HMI tags "2920RS001A01T02"
   "2920RS001A01T02.MSW" : 52809b66-421d-457f-8884-6f7a49d4e247 AT %DB5053.DBX18.0, 500 ms
   "2920RS001A01T02.DefaultText" : TextRef, internal   // Заголовок POPUP окна. При експорте из ECS через скрипт заполняется автоматически, если теги копируются в ручную то требуется в ручную задатать свойство Start Value
   "2920RS001A01T02.BlockInfo" : Array [0..2] of Int AT %DB5053.DBX38.0, 500 ms
   "2920RS001A01T02.StatusWork" : Int AT %DB5053.DBW242, 500 ms
   "2920RS001A01T02.FP_PARAM.DampingTime" : Int AT %DB5053.DBW50, 500 ms
   "2920RS001A01T02.FP_PARAM.Force_Value" : Real AT %DB5053.DBD52, 500 ms
   "2920RS001A01T02.FP_PARAM.Scale_Min" : Real AT %DB5053.DBD56, 500 ms
   "2920RS001A01T02.FP_PARAM.Scale_Max" : Real AT %DB5053.DBD60, 500 ms
   "2920RS001A01T02.FP_PARAM.Gradient" : Real AT %DB5053.DBD64, 500 ms
   "2920RS001A01T02.FP_PARAM.Grad_Pos" : Real AT %DB5053.DBD68, 500 ms
   "2920RS001A01T02.FP_PARAM.Grad_Neg" : Real AT %DB5053.DBD72, 500 ms
   "2920RS001A01T02.FP_PARAM.Grad_X" : Real AT %DB5053.DBD76, 500 ms
   "2920RS001A01T02.FP_PARAM.Gradient_Time_Pre" : Int AT %DB5053.DBW80, 500 ms
   "2920RS001A01T02.FP_PARAM.Gradient_Time_ACC" : Int AT %DB5053.DBW82, 500 ms
   "2920RS001A01T02.FP_PARAM.Alarm_Hyst" : Real AT %DB5053.DBD84, 500 ms
   "2920RS001A01T02.FP_PARAM.AlarmLimit_H3" : Real AT %DB5053.DBD88, 500 ms
   "2920RS001A01T02.FP_PARAM.AlarmLimit_H2" : Real AT %DB5053.DBD92, 500 ms
   "2920RS001A01T02.FP_PARAM.AlarmLimit_H1" : Real AT %DB5053.DBD96, 500 ms
   "2920RS001A01T02.FP_PARAM.AlarmLimit_L1" : Real AT %DB5053.DBD100, 500 ms
   "2920RS001A01T02.FP_PARAM.AlarmLimit_L2" : Real AT %DB5053.DBD104, 500 ms
   "2920RS001A01T02.FP_PARAM.AlarmLimit_L3" : Real AT %DB5053.DBD108, 500 ms
   "2920RS001A01T02.FP_PARAM.AlarmDelay_H3_Pre" : Int AT %DB5053.DBW112, 500 ms
   "2920RS001A01T02.FP_PARAM.AlarmDelay_H3_Acc" : Int AT %DB5053.DBW114, 500 ms
   "2920RS001A01T02.FP_PARAM.AlarmDelay_H2_Pre" : Int AT %DB5053.DBW116, 500 ms
   "2920RS001A01T02.FP_PARAM.AlarmDelay_H2_Acc" : Int AT %DB5053.DBW118, 500 ms
   "2920RS001A01T02.FP_PARAM.AlarmDelay_H1_Pre" : Int AT %DB5053.DBW120, 500 ms
   "2920RS001A01T02.FP_PARAM.AlarmDelay_H1_Acc" : Int AT %DB5053.DBW122, 500 ms
   "2920RS001A01T02.FP_PARAM.AlarmDelay_L1_Pre" : Int AT %DB5053.DBW124, 500 ms
   "2920RS001A01T02.FP_PARAM.AlarmDelay_L1_Acc" : Int AT %DB5053.DBW126, 500 ms
   "2920RS001A01T02.FP_PARAM.AlarmDelay_L2_Pre" : Int AT %DB5053.DBW128, 500 ms
   "2920RS001A01T02.FP_PARAM.AlarmDelay_L2_Acc" : Int AT %DB5053.DBW130, 500 ms
   "2920RS001A01T02.FP_PARAM.AlarmDelay_L3_Pre" : Int AT %DB5053.DBW132, 500 ms
   "2920RS001A01T02.FP_PARAM.AlarmDelay_L3_Acc" : Int AT %DB5053.DBW134, 500 ms
   "2920RS001A01T02.FP_PARAM.OpenLoopDelay_Pre" : Int AT %DB5053.DBW136, 500 ms
   "2920RS001A01T02.FP_PARAM.OpenLoopDelay_Acc" : Int AT %DB5053.DBW138, 500 ms
   "2920RS001A01T02.FP_PARAM.OverRangeDelay_Pre" : Int AT %DB5053.DBW140, 500 ms
   "2920RS001A01T02.FP_PARAM.OverRangeDelay_Acc" : Int AT %DB5053.DBW142, 500 ms
   "2920RS001A01T02.FP_PARAM.AuxLimit_H2_Value" : Real AT %DB5053.DBD144, 500 ms
   "2920RS001A01T02.FP_PARAM.AuxLimit_H1_Value" : Real AT %DB5053.DBD148, 500 ms
   "2920RS001A01T02.FP_PARAM.AuxLimit_L2_Value" : Real AT %DB5053.DBD152, 500 ms
   "2920RS001A01T02.FP_PARAM.AuxLimit_L1_Value" : Real AT %DB5053.DBD156, 500 ms
   "2920RS001A01T02.Unit" : TextRef, internal   // Еденицы измерения При експорте из ECS через скрипт заполняется автоматически, если теги копируются в ручную то требуется задатать свойство Text
   "2920RS001A01T02.Decimals" : TextRef, internal   // Формат отображения При експорте из ECS через скрипт, заполняется автоматически. Если теги копируются в ручную то требуется задатать свойство Text s999999.9
   "2920RS001A01T02.FP_EN.Square" : Bool AT %DB5053.DBX46.0, 500 ms
   "2920RS001A01T02.FP_EN.SquareRoot" : Bool AT %DB5053.DBX46.1, 500 ms
   "2920RS001A01T02.FP_EN.ParentSupress" : Bool AT %DB5053.DBX46.2, 500 ms
   "2920RS001A01T02.FP_EN.ParentSupressUnit" : Bool AT %DB5053.DBX46.3, 500 ms
   "2920RS001A01T02.FP_EN.Force" : Bool AT %DB5053.DBX46.4, 500 ms
   "2920RS001A01T02.FP_EN.Damping" : Bool AT %DB5053.DBX46.5, 500 ms
   "2920RS001A01T02.FP_EN.Gradient_Pos" : Bool AT %DB5053.DBX46.6, 500 ms
   "2920RS001A01T02.FP_EN.Gradient_Neg" : Bool AT %DB5053.DBX46.7, 500 ms
   "2920RS001A01T02.FP_EN.Hysteresis" : Bool AT %DB5053.DBX47.0, 500 ms
   "2920RS001A01T02.FP_EN.Alarm_H3" : Bool AT %DB5053.DBX47.1, 500 ms
   "2920RS001A01T02.FP_EN.Alarm_H2" : Bool AT %DB5053.DBX47.2, 500 ms
   "2920RS001A01T02.FP_EN.Alarm_H1" : Bool AT %DB5053.DBX47.3, 500 ms
   "2920RS001A01T02.FP_EN.Alarm_L1" : Bool AT %DB5053.DBX47.4, 500 ms
   "2920RS001A01T02.FP_EN.Alarm_L2" : Bool AT %DB5053.DBX47.5, 500 ms
   "2920RS001A01T02.FP_EN.Alarm_L3" : Bool AT %DB5053.DBX47.6, 500 ms
   "2920RS001A01T02.FP_EN.AlarmDelay_H3" : Bool AT %DB5053.DBX47.7, 500 ms
   "2920RS001A01T02.FP_EN.AlarmDelay_H2" : Bool AT %DB5053.DBX48.0, 500 ms
   "2920RS001A01T02.FP_EN.AlarmDelay_H1" : Bool AT %DB5053.DBX48.1, 500 ms
   "2920RS001A01T02.FP_EN.AlarmDelay_L1" : Bool AT %DB5053.DBX48.2, 500 ms
   "2920RS001A01T02.FP_EN.AlarmDelay_L2" : Bool AT %DB5053.DBX48.3, 500 ms
   "2920RS001A01T02.FP_EN.AlarmDelay_L3" : Bool AT %DB5053.DBX48.4, 500 ms
   "2920RS001A01T02.FP_EN.ROC_Warn" : Bool AT %DB5053.DBX48.5, 500 ms
   "2920RS001A01T02.FP_EN.U_Range_Warn" : Bool AT %DB5053.DBX48.6, 500 ms
   "2920RS001A01T02.FP_EN.O_Range_Warn" : Bool AT %DB5053.DBX48.7, 500 ms
   "2920RS001A01T02.trend_tag_name" : TextRef, internal   // Еденицы измерения При експорте из ECS через скрипт - заполняется автоматически, если теги копируются в ручную то требуется задатать свойство Text - имя тега для тренда
   "2920RS001A01T02.DQ.AL_H3" : Bool AT %DB5053.DBX16.0, 500 ms
   "2920RS001A01T02.DQ.AL_H2" : Bool AT %DB5053.DBX16.1, 500 ms
   "2920RS001A01T02.DQ.AL_H1" : Bool AT %DB5053.DBX16.2, 500 ms
   "2920RS001A01T02.DQ.AL_L1" : Bool AT %DB5053.DBX16.3, 500 ms
   "2920RS001A01T02.DQ.AL_L2" : Bool AT %DB5053.DBX16.4, 500 ms
   "2920RS001A01T02.DQ.AL_L3" : Bool AT %DB5053.DBX16.5, 500 ms
   "2920RS001A01T02.DQ.SIG_OK" : Bool AT %DB5053.DBX16.6, 500 ms
   "2920RS001A01T02.DQ.LIM_H2" : Bool AT %DB5053.DBX16.7, 500 ms
   "2920RS001A01T02.DQ.LIM_H1" : Bool AT %DB5053.DBX17.0, 500 ms
   "2920RS001A01T02.DQ.LIM_L1" : Bool AT %DB5053.DBX17.1, 500 ms
   "2920RS001A01T02.DQ.LIM_L2" : Bool AT %DB5053.DBX17.2, 500 ms
   "2920RS001A01T02.DQ.GR_P" : Bool AT %DB5053.DBX17.3, 500 ms
   "2920RS001A01T02.DQ.GR_N" : Bool AT %DB5053.DBX17.4, 500 ms
   "2920RS001A01T02.I.IN" : Real AT %DB5053.DBD2, 500 ms
   "2920RS001A01T02.I.SIG_TYPE" : Int AT %DB5053.DBW0, 500 ms
   "2920RS001A01T02.I.FI_BUS" : Byte AT %DB5053.DBB6, 500 ms
   "2920RS001A01T02.DI.U_RANGE" : Bool AT %DB5053.DBX7.0, 500 ms
   "2920RS001A01T02.DI.O_RANGE" : Bool AT %DB5053.DBX7.1, 500 ms
   "2920RS001A01T02.DI.SIG_FAULT" : Bool AT %DB5053.DBX7.2, 500 ms
   "2920RS001A01T02.DI.EnConfig" : Bool AT %DB5053.DBX7.3, 500 ms
   "2920RS001A01T02.DI.AEN" : Bool AT %DB5053.DBX7.4, 500 ms
   "2920RS001A01T02.DI.AL_SUPR" : Bool AT %DB5053.DBX7.5, 500 ms
   "2920RS001A01T02.Q.PV_NORM" : Real AT %DB5053.DBD8, 500 ms
   "2920RS001A01T02.Q.PV_SCAL" : Real AT %DB5053.DBD12, 500 ms
   "2920RS001A01T02.ParentInfo" : TextRef, internal   // Имя родителя для попап окна, вкладка инфо. При експорте из ECS через скрипт заполняется автоматически, если теги копируются в ручную то требуется в ручную задатать свойство Start Value

HMI tags "2920RS001A01T03"
   "2920RS001A01T03.MSW" : 52809b66-421d-457f-8884-6f7a49d4e247 AT %DB5054.DBX18.0, 500 ms
   "2920RS001A01T03.DefaultText" : TextRef, internal   // Заголовок POPUP окна. При експорте из ECS через скрипт заполняется автоматически, если теги копируются в ручную то требуется в ручную задатать свойство Start Value
   "2920RS001A01T03.BlockInfo" : Array [0..2] of Int AT %DB5054.DBX38.0, 500 ms
   "2920RS001A01T03.StatusWork" : Int AT %DB5054.DBW242, 500 ms
   "2920RS001A01T03.FP_PARAM.DampingTime" : Int AT %DB5054.DBW50, 500 ms
   "2920RS001A01T03.FP_PARAM.Force_Value" : Real AT %DB5054.DBD52, 500 ms
   "2920RS001A01T03.FP_PARAM.Scale_Min" : Real AT %DB5054.DBD56, 500 ms
   "2920RS001A01T03.FP_PARAM.Scale_Max" : Real AT %DB5054.DBD60, 500 ms
   "2920RS001A01T03.FP_PARAM.Gradient" : Real AT %DB5054.DBD64, 500 ms
   "2920RS001A01T03.FP_PARAM.Grad_Pos" : Real AT %DB5054.DBD68, 500 ms
   "2920RS001A01T03.FP_PARAM.Grad_Neg" : Real AT %DB5054.DBD72, 500 ms
   "2920RS001A01T03.FP_PARAM.Grad_X" : Real AT %DB5054.DBD76, 500 ms
   "2920RS001A01T03.FP_PARAM.Gradient_Time_Pre" : Int AT %DB5054.DBW80, 500 ms
   "2920RS001A01T03.FP_PARAM.Gradient_Time_ACC" : Int AT %DB5054.DBW82, 500 ms
   "2920RS001A01T03.FP_PARAM.Alarm_Hyst" : Real AT %DB5054.DBD84, 500 ms
   "2920RS001A01T03.FP_PARAM.AlarmLimit_H3" : Real AT %DB5054.DBD88, 500 ms
   "2920RS001A01T03.FP_PARAM.AlarmLimit_H2" : Real AT %DB5054.DBD92, 500 ms
   "2920RS001A01T03.FP_PARAM.AlarmLimit_H1" : Real AT %DB5054.DBD96, 500 ms
   "2920RS001A01T03.FP_PARAM.AlarmLimit_L1" : Real AT %DB5054.DBD100, 500 ms
   "2920RS001A01T03.FP_PARAM.AlarmLimit_L2" : Real AT %DB5054.DBD104, 500 ms
   "2920RS001A01T03.FP_PARAM.AlarmLimit_L3" : Real AT %DB5054.DBD108, 500 ms
   "2920RS001A01T03.FP_PARAM.AlarmDelay_H3_Pre" : Int AT %DB5054.DBW112, 500 ms
   "2920RS001A01T03.FP_PARAM.AlarmDelay_H3_Acc" : Int AT %DB5054.DBW114, 500 ms
   "2920RS001A01T03.FP_PARAM.AlarmDelay_H2_Pre" : Int AT %DB5054.DBW116, 500 ms
   "2920RS001A01T03.FP_PARAM.AlarmDelay_H2_Acc" : Int AT %DB5054.DBW118, 500 ms
   "2920RS001A01T03.FP_PARAM.AlarmDelay_H1_Pre" : Int AT %DB5054.DBW120, 500 ms
   "2920RS001A01T03.FP_PARAM.AlarmDelay_H1_Acc" : Int AT %DB5054.DBW122, 500 ms
   "2920RS001A01T03.FP_PARAM.AlarmDelay_L1_Pre" : Int AT %DB5054.DBW124, 500 ms
   "2920RS001A01T03.FP_PARAM.AlarmDelay_L1_Acc" : Int AT %DB5054.DBW126, 500 ms
   "2920RS001A01T03.FP_PARAM.AlarmDelay_L2_Pre" : Int AT %DB5054.DBW128, 500 ms
   "2920RS001A01T03.FP_PARAM.AlarmDelay_L2_Acc" : Int AT %DB5054.DBW130, 500 ms
   "2920RS001A01T03.FP_PARAM.AlarmDelay_L3_Pre" : Int AT %DB5054.DBW132, 500 ms
   "2920RS001A01T03.FP_PARAM.AlarmDelay_L3_Acc" : Int AT %DB5054.DBW134, 500 ms
   "2920RS001A01T03.FP_PARAM.OpenLoopDelay_Pre" : Int AT %DB5054.DBW136, 500 ms
   "2920RS001A01T03.FP_PARAM.OpenLoopDelay_Acc" : Int AT %DB5054.DBW138, 500 ms
   "2920RS001A01T03.FP_PARAM.OverRangeDelay_Pre" : Int AT %DB5054.DBW140, 500 ms
   "2920RS001A01T03.FP_PARAM.OverRangeDelay_Acc" : Int AT %DB5054.DBW142, 500 ms
   "2920RS001A01T03.FP_PARAM.AuxLimit_H2_Value" : Real AT %DB5054.DBD144, 500 ms
   "2920RS001A01T03.FP_PARAM.AuxLimit_H1_Value" : Real AT %DB5054.DBD148, 500 ms
   "2920RS001A01T03.FP_PARAM.AuxLimit_L2_Value" : Real AT %DB5054.DBD152, 500 ms
   "2920RS001A01T03.FP_PARAM.AuxLimit_L1_Value" : Real AT %DB5054.DBD156, 500 ms
   "2920RS001A01T03.Unit" : TextRef, internal   // Еденицы измерения При експорте из ECS через скрипт заполняется автоматически, если теги копируются в ручную то требуется задатать свойство Text
   "2920RS001A01T03.Decimals" : TextRef, internal   // Формат отображения При експорте из ECS через скрипт, заполняется автоматически. Если теги копируются в ручную то требуется задатать свойство Text s999999.9
   "2920RS001A01T03.FP_EN.Square" : Bool AT %DB5054.DBX46.0, 500 ms
   "2920RS001A01T03.FP_EN.SquareRoot" : Bool AT %DB5054.DBX46.1, 500 ms
   "2920RS001A01T03.FP_EN.ParentSupress" : Bool AT %DB5054.DBX46.2, 500 ms
   "2920RS001A01T03.FP_EN.ParentSupressUnit" : Bool AT %DB5054.DBX46.3, 500 ms
   "2920RS001A01T03.FP_EN.Force" : Bool AT %DB5054.DBX46.4, 500 ms
   "2920RS001A01T03.FP_EN.Damping" : Bool AT %DB5054.DBX46.5, 500 ms
   "2920RS001A01T03.FP_EN.Gradient_Pos" : Bool AT %DB5054.DBX46.6, 500 ms
   "2920RS001A01T03.FP_EN.Gradient_Neg" : Bool AT %DB5054.DBX46.7, 500 ms
   "2920RS001A01T03.FP_EN.Hysteresis" : Bool AT %DB5054.DBX47.0, 500 ms
   "2920RS001A01T03.FP_EN.Alarm_H3" : Bool AT %DB5054.DBX47.1, 500 ms
   "2920RS001A01T03.FP_EN.Alarm_H2" : Bool AT %DB5054.DBX47.2, 500 ms
   "2920RS001A01T03.FP_EN.Alarm_H1" : Bool AT %DB5054.DBX47.3, 500 ms
   "2920RS001A01T03.FP_EN.Alarm_L1" : Bool AT %DB5054.DBX47.4, 500 ms
   "2920RS001A01T03.FP_EN.Alarm_L2" : Bool AT %DB5054.DBX47.5, 500 ms
   "2920RS001A01T03.FP_EN.Alarm_L3" : Bool AT %DB5054.DBX47.6, 500 ms
   "2920RS001A01T03.FP_EN.AlarmDelay_H3" : Bool AT %DB5054.DBX47.7, 500 ms
   "2920RS001A01T03.FP_EN.AlarmDelay_H2" : Bool AT %DB5054.DBX48.0, 500 ms
   "2920RS001A01T03.FP_EN.AlarmDelay_H1" : Bool AT %DB5054.DBX48.1, 500 ms
   "2920RS001A01T03.FP_EN.AlarmDelay_L1" : Bool AT %DB5054.DBX48.2, 500 ms
   "2920RS001A01T03.FP_EN.AlarmDelay_L2" : Bool AT %DB5054.DBX48.3, 500 ms
   "2920RS001A01T03.FP_EN.AlarmDelay_L3" : Bool AT %DB5054.DBX48.4, 500 ms
   "2920RS001A01T03.FP_EN.ROC_Warn" : Bool AT %DB5054.DBX48.5, 500 ms
   "2920RS001A01T03.FP_EN.U_Range_Warn" : Bool AT %DB5054.DBX48.6, 500 ms
   "2920RS001A01T03.FP_EN.O_Range_Warn" : Bool AT %DB5054.DBX48.7, 500 ms
   "2920RS001A01T03.trend_tag_name" : TextRef, internal   // Еденицы измерения При експорте из ECS через скрипт - заполняется автоматически, если теги копируются в ручную то требуется задатать свойство Text - имя тега для тренда
   "2920RS001A01T03.DQ.AL_H3" : Bool AT %DB5054.DBX16.0, 500 ms
   "2920RS001A01T03.DQ.AL_H2" : Bool AT %DB5054.DBX16.1, 500 ms
   "2920RS001A01T03.DQ.AL_H1" : Bool AT %DB5054.DBX16.2, 500 ms
   "2920RS001A01T03.DQ.AL_L1" : Bool AT %DB5054.DBX16.3, 500 ms
   "2920RS001A01T03.DQ.AL_L2" : Bool AT %DB5054.DBX16.4, 500 ms
   "2920RS001A01T03.DQ.AL_L3" : Bool AT %DB5054.DBX16.5, 500 ms
   "2920RS001A01T03.DQ.SIG_OK" : Bool AT %DB5054.DBX16.6, 500 ms
   "2920RS001A01T03.DQ.LIM_H2" : Bool AT %DB5054.DBX16.7, 500 ms
   "2920RS001A01T03.DQ.LIM_H1" : Bool AT %DB5054.DBX17.0, 500 ms
   "2920RS001A01T03.DQ.LIM_L1" : Bool AT %DB5054.DBX17.1, 500 ms
   "2920RS001A01T03.DQ.LIM_L2" : Bool AT %DB5054.DBX17.2, 500 ms
   "2920RS001A01T03.DQ.GR_P" : Bool AT %DB5054.DBX17.3, 500 ms
   "2920RS001A01T03.DQ.GR_N" : Bool AT %DB5054.DBX17.4, 500 ms
   "2920RS001A01T03.I.IN" : Real AT %DB5054.DBD2, 500 ms
   "2920RS001A01T03.I.SIG_TYPE" : Int AT %DB5054.DBW0, 500 ms
   "2920RS001A01T03.I.FI_BUS" : Byte AT %DB5054.DBB6, 500 ms
   "2920RS001A01T03.DI.U_RANGE" : Bool AT %DB5054.DBX7.0, 500 ms
   "2920RS001A01T03.DI.O_RANGE" : Bool AT %DB5054.DBX7.1, 500 ms
   "2920RS001A01T03.DI.SIG_FAULT" : Bool AT %DB5054.DBX7.2, 500 ms
   "2920RS001A01T03.DI.EnConfig" : Bool AT %DB5054.DBX7.3, 500 ms
   "2920RS001A01T03.DI.AEN" : Bool AT %DB5054.DBX7.4, 500 ms
   "2920RS001A01T03.DI.AL_SUPR" : Bool AT %DB5054.DBX7.5, 500 ms
   "2920RS001A01T03.Q.PV_NORM" : Real AT %DB5054.DBD8, 500 ms
   "2920RS001A01T03.Q.PV_SCAL" : Real AT %DB5054.DBD12, 500 ms
   "2920RS001A01T03.ParentInfo" : TextRef, internal   // Имя родителя для попап окна, вкладка инфо. При експорте из ECS через скрипт заполняется автоматически, если теги копируются в ручную то требуется в ручную задатать свойство Start Value

HMI tags "2920RS001A01T04"
   "2920RS001A01T04.MSW" : 52809b66-421d-457f-8884-6f7a49d4e247 AT %DB5055.DBX18.0, 500 ms
   "2920RS001A01T04.DefaultText" : TextRef, internal   // Заголовок POPUP окна. При експорте из ECS через скрипт заполняется автоматически, если теги копируются в ручную то требуется в ручную задатать свойство Start Value
   "2920RS001A01T04.BlockInfo" : Array [0..2] of Int AT %DB5055.DBX38.0, 500 ms
   "2920RS001A01T04.StatusWork" : Int AT %DB5055.DBW242, 500 ms
   "2920RS001A01T04.FP_PARAM.DampingTime" : Int AT %DB5055.DBW50, 500 ms
   "2920RS001A01T04.FP_PARAM.Force_Value" : Real AT %DB5055.DBD52, 500 ms
   "2920RS001A01T04.FP_PARAM.Scale_Min" : Real AT %DB5055.DBD56, 500 ms
   "2920RS001A01T04.FP_PARAM.Scale_Max" : Real AT %DB5055.DBD60, 500 ms
   "2920RS001A01T04.FP_PARAM.Gradient" : Real AT %DB5055.DBD64, 500 ms
   "2920RS001A01T04.FP_PARAM.Grad_Pos" : Real AT %DB5055.DBD68, 500 ms
   "2920RS001A01T04.FP_PARAM.Grad_Neg" : Real AT %DB5055.DBD72, 500 ms
   "2920RS001A01T04.FP_PARAM.Grad_X" : Real AT %DB5055.DBD76, 500 ms
   "2920RS001A01T04.FP_PARAM.Gradient_Time_Pre" : Int AT %DB5055.DBW80, 500 ms
   "2920RS001A01T04.FP_PARAM.Gradient_Time_ACC" : Int AT %DB5055.DBW82, 500 ms
   "2920RS001A01T04.FP_PARAM.Alarm_Hyst" : Real AT %DB5055.DBD84, 500 ms
   "2920RS001A01T04.FP_PARAM.AlarmLimit_H3" : Real AT %DB5055.DBD88, 500 ms
   "2920RS001A01T04.FP_PARAM.AlarmLimit_H2" : Real AT %DB5055.DBD92, 500 ms
   "2920RS001A01T04.FP_PARAM.AlarmLimit_H1" : Real AT %DB5055.DBD96, 500 ms
   "2920RS001A01T04.FP_PARAM.AlarmLimit_L1" : Real AT %DB5055.DBD100, 500 ms
   "2920RS001A01T04.FP_PARAM.AlarmLimit_L2" : Real AT %DB5055.DBD104, 500 ms
   "2920RS001A01T04.FP_PARAM.AlarmLimit_L3" : Real AT %DB5055.DBD108, 500 ms
   "2920RS001A01T04.FP_PARAM.AlarmDelay_H3_Pre" : Int AT %DB5055.DBW112, 500 ms
   "2920RS001A01T04.FP_PARAM.AlarmDelay_H3_Acc" : Int AT %DB5055.DBW114, 500 ms
   "2920RS001A01T04.FP_PARAM.AlarmDelay_H2_Pre" : Int AT %DB5055.DBW116, 500 ms
   "2920RS001A01T04.FP_PARAM.AlarmDelay_H2_Acc" : Int AT %DB5055.DBW118, 500 ms
   "2920RS001A01T04.FP_PARAM.AlarmDelay_H1_Pre" : Int AT %DB5055.DBW120, 500 ms
   "2920RS001A01T04.FP_PARAM.AlarmDelay_H1_Acc" : Int AT %DB5055.DBW122, 500 ms
   "2920RS001A01T04.FP_PARAM.AlarmDelay_L1_Pre" : Int AT %DB5055.DBW124, 500 ms
   "2920RS001A01T04.FP_PARAM.AlarmDelay_L1_Acc" : Int AT %DB5055.DBW126, 500 ms
   "2920RS001A01T04.FP_PARAM.AlarmDelay_L2_Pre" : Int AT %DB5055.DBW128, 500 ms
   "2920RS001A01T04.FP_PARAM.AlarmDelay_L2_Acc" : Int AT %DB5055.DBW130, 500 ms
   "2920RS001A01T04.FP_PARAM.AlarmDelay_L3_Pre" : Int AT %DB5055.DBW132, 500 ms
   "2920RS001A01T04.FP_PARAM.AlarmDelay_L3_Acc" : Int AT %DB5055.DBW134, 500 ms
   "2920RS001A01T04.FP_PARAM.OpenLoopDelay_Pre" : Int AT %DB5055.DBW136, 500 ms
   "2920RS001A01T04.FP_PARAM.OpenLoopDelay_Acc" : Int AT %DB5055.DBW138, 500 ms
   "2920RS001A01T04.FP_PARAM.OverRangeDelay_Pre" : Int AT %DB5055.DBW140, 500 ms
   "2920RS001A01T04.FP_PARAM.OverRangeDelay_Acc" : Int AT %DB5055.DBW142, 500 ms
   "2920RS001A01T04.FP_PARAM.AuxLimit_H2_Value" : Real AT %DB5055.DBD144, 500 ms
   "2920RS001A01T04.FP_PARAM.AuxLimit_H1_Value" : Real AT %DB5055.DBD148, 500 ms
   "2920RS001A01T04.FP_PARAM.AuxLimit_L2_Value" : Real AT %DB5055.DBD152, 500 ms
   "2920RS001A01T04.FP_PARAM.AuxLimit_L1_Value" : Real AT %DB5055.DBD156, 500 ms
   "2920RS001A01T04.Unit" : TextRef, internal   // Еденицы измерения При експорте из ECS через скрипт заполняется автоматически, если теги копируются в ручную то требуется задатать свойство Text
   "2920RS001A01T04.Decimals" : TextRef, internal   // Формат отображения При експорте из ECS через скрипт, заполняется автоматически. Если теги копируются в ручную то требуется задатать свойство Text s999999.9
   "2920RS001A01T04.FP_EN.Square" : Bool AT %DB5055.DBX46.0, 500 ms
   "2920RS001A01T04.FP_EN.SquareRoot" : Bool AT %DB5055.DBX46.1, 500 ms
   "2920RS001A01T04.FP_EN.ParentSupress" : Bool AT %DB5055.DBX46.2, 500 ms
   "2920RS001A01T04.FP_EN.ParentSupressUnit" : Bool AT %DB5055.DBX46.3, 500 ms
   "2920RS001A01T04.FP_EN.Force" : Bool AT %DB5055.DBX46.4, 500 ms
   "2920RS001A01T04.FP_EN.Damping" : Bool AT %DB5055.DBX46.5, 500 ms
   "2920RS001A01T04.FP_EN.Gradient_Pos" : Bool AT %DB5055.DBX46.6, 500 ms
   "2920RS001A01T04.FP_EN.Gradient_Neg" : Bool AT %DB5055.DBX46.7, 500 ms
   "2920RS001A01T04.FP_EN.Hysteresis" : Bool AT %DB5055.DBX47.0, 500 ms
   "2920RS001A01T04.FP_EN.Alarm_H3" : Bool AT %DB5055.DBX47.1, 500 ms
   "2920RS001A01T04.FP_EN.Alarm_H2" : Bool AT %DB5055.DBX47.2, 500 ms
   "2920RS001A01T04.FP_EN.Alarm_H1" : Bool AT %DB5055.DBX47.3, 500 ms
   "2920RS001A01T04.FP_EN.Alarm_L1" : Bool AT %DB5055.DBX47.4, 500 ms
   "2920RS001A01T04.FP_EN.Alarm_L2" : Bool AT %DB5055.DBX47.5, 500 ms
   "2920RS001A01T04.FP_EN.Alarm_L3" : Bool AT %DB5055.DBX47.6, 500 ms
   "2920RS001A01T04.FP_EN.AlarmDelay_H3" : Bool AT %DB5055.DBX47.7, 500 ms
   "2920RS001A01T04.FP_EN.AlarmDelay_H2" : Bool AT %DB5055.DBX48.0, 500 ms
   "2920RS001A01T04.FP_EN.AlarmDelay_H1" : Bool AT %DB5055.DBX48.1, 500 ms
   "2920RS001A01T04.FP_EN.AlarmDelay_L1" : Bool AT %DB5055.DBX48.2, 500 ms
   "2920RS001A01T04.FP_EN.AlarmDelay_L2" : Bool AT %DB5055.DBX48.3, 500 ms
   "2920RS001A01T04.FP_EN.AlarmDelay_L3" : Bool AT %DB5055.DBX48.4, 500 ms
   "2920RS001A01T04.FP_EN.ROC_Warn" : Bool AT %DB5055.DBX48.5, 500 ms
   "2920RS001A01T04.FP_EN.U_Range_Warn" : Bool AT %DB5055.DBX48.6, 500 ms
   "2920RS001A01T04.FP_EN.O_Range_Warn" : Bool AT %DB5055.DBX48.7, 500 ms
   "2920RS001A01T04.trend_tag_name" : TextRef, internal   // Еденицы измерения При експорте из ECS через скрипт - заполняется автоматически, если теги копируются в ручную то требуется задатать свойство Text - имя тега для тренда
   "2920RS001A01T04.DQ.AL_H3" : Bool AT %DB5055.DBX16.0, 500 ms
   "2920RS001A01T04.DQ.AL_H2" : Bool AT %DB5055.DBX16.1, 500 ms
   "2920RS001A01T04.DQ.AL_H1" : Bool AT %DB5055.DBX16.2, 500 ms
   "2920RS001A01T04.DQ.AL_L1" : Bool AT %DB5055.DBX16.3, 500 ms
   "2920RS001A01T04.DQ.AL_L2" : Bool AT %DB5055.DBX16.4, 500 ms
   "2920RS001A01T04.DQ.AL_L3" : Bool AT %DB5055.DBX16.5, 500 ms
   "2920RS001A01T04.DQ.SIG_OK" : Bool AT %DB5055.DBX16.6, 500 ms
   "2920RS001A01T04.DQ.LIM_H2" : Bool AT %DB5055.DBX16.7, 500 ms
   "2920RS001A01T04.DQ.LIM_H1" : Bool AT %DB5055.DBX17.0, 500 ms
   "2920RS001A01T04.DQ.LIM_L1" : Bool AT %DB5055.DBX17.1, 500 ms
   "2920RS001A01T04.DQ.LIM_L2" : Bool AT %DB5055.DBX17.2, 500 ms
   "2920RS001A01T04.DQ.GR_P" : Bool AT %DB5055.DBX17.3, 500 ms
   "2920RS001A01T04.DQ.GR_N" : Bool AT %DB5055.DBX17.4, 500 ms
   "2920RS001A01T04.I.IN" : Real AT %DB5055.DBD2, 500 ms
   "2920RS001A01T04.I.SIG_TYPE" : Int AT %DB5055.DBW0, 500 ms
   "2920RS001A01T04.I.FI_BUS" : Byte AT %DB5055.DBB6, 500 ms
   "2920RS001A01T04.DI.U_RANGE" : Bool AT %DB5055.DBX7.0, 500 ms
   "2920RS001A01T04.DI.O_RANGE" : Bool AT %DB5055.DBX7.1, 500 ms
   "2920RS001A01T04.DI.SIG_FAULT" : Bool AT %DB5055.DBX7.2, 500 ms
   "2920RS001A01T04.DI.EnConfig" : Bool AT %DB5055.DBX7.3, 500 ms
   "2920RS001A01T04.DI.AEN" : Bool AT %DB5055.DBX7.4, 500 ms
   "2920RS001A01T04.DI.AL_SUPR" : Bool AT %DB5055.DBX7.5, 500 ms
   "2920RS001A01T04.Q.PV_NORM" : Real AT %DB5055.DBD8, 500 ms
   "2920RS001A01T04.Q.PV_SCAL" : Real AT %DB5055.DBD12, 500 ms
   "2920RS001A01T04.ParentInfo" : TextRef, internal   // Имя родителя для попап окна, вкладка инфо. При експорте из ECS через скрипт заполняется автоматически, если теги копируются в ручную то требуется в ручную задатать свойство Start Value

HMI tags "2920RS001A01T05"
   "2920RS001A01T05.MSW" : 52809b66-421d-457f-8884-6f7a49d4e247 AT %DB5056.DBX18.0, 500 ms
   "2920RS001A01T05.DefaultText" : TextRef, internal   // Заголовок POPUP окна. При експорте из ECS через скрипт заполняется автоматически, если теги копируются в ручную то требуется в ручную задатать свойство Start Value
   "2920RS001A01T05.BlockInfo" : Array [0..2] of Int AT %DB5056.DBX38.0, 500 ms
   "2920RS001A01T05.StatusWork" : Int AT %DB5056.DBW242, 500 ms
   "2920RS001A01T05.FP_PARAM.DampingTime" : Int AT %DB5056.DBW50, 500 ms
   "2920RS001A01T05.FP_PARAM.Force_Value" : Real AT %DB5056.DBD52, 500 ms
   "2920RS001A01T05.FP_PARAM.Scale_Min" : Real AT %DB5056.DBD56, 500 ms
   "2920RS001A01T05.FP_PARAM.Scale_Max" : Real AT %DB5056.DBD60, 500 ms
   "2920RS001A01T05.FP_PARAM.Gradient" : Real AT %DB5056.DBD64, 500 ms
   "2920RS001A01T05.FP_PARAM.Grad_Pos" : Real AT %DB5056.DBD68, 500 ms
   "2920RS001A01T05.FP_PARAM.Grad_Neg" : Real AT %DB5056.DBD72, 500 ms
   "2920RS001A01T05.FP_PARAM.Grad_X" : Real AT %DB5056.DBD76, 500 ms
   "2920RS001A01T05.FP_PARAM.Gradient_Time_Pre" : Int AT %DB5056.DBW80, 500 ms
   "2920RS001A01T05.FP_PARAM.Gradient_Time_ACC" : Int AT %DB5056.DBW82, 500 ms
   "2920RS001A01T05.FP_PARAM.Alarm_Hyst" : Real AT %DB5056.DBD84, 500 ms
   "2920RS001A01T05.FP_PARAM.AlarmLimit_H3" : Real AT %DB5056.DBD88, 500 ms
   "2920RS001A01T05.FP_PARAM.AlarmLimit_H2" : Real AT %DB5056.DBD92, 500 ms
   "2920RS001A01T05.FP_PARAM.AlarmLimit_H1" : Real AT %DB5056.DBD96, 500 ms
   "2920RS001A01T05.FP_PARAM.AlarmLimit_L1" : Real AT %DB5056.DBD100, 500 ms
   "2920RS001A01T05.FP_PARAM.AlarmLimit_L2" : Real AT %DB5056.DBD104, 500 ms
   "2920RS001A01T05.FP_PARAM.AlarmLimit_L3" : Real AT %DB5056.DBD108, 500 ms
   "2920RS001A01T05.FP_PARAM.AlarmDelay_H3_Pre" : Int AT %DB5056.DBW112, 500 ms
   "2920RS001A01T05.FP_PARAM.AlarmDelay_H3_Acc" : Int AT %DB5056.DBW114, 500 ms
   "2920RS001A01T05.FP_PARAM.AlarmDelay_H2_Pre" : Int AT %DB5056.DBW116, 500 ms
   "2920RS001A01T05.FP_PARAM.AlarmDelay_H2_Acc" : Int AT %DB5056.DBW118, 500 ms
   "2920RS001A01T05.FP_PARAM.AlarmDelay_H1_Pre" : Int AT %DB5056.DBW120, 500 ms
   "2920RS001A01T05.FP_PARAM.AlarmDelay_H1_Acc" : Int AT %DB5056.DBW122, 500 ms
   "2920RS001A01T05.FP_PARAM.AlarmDelay_L1_Pre" : Int AT %DB5056.DBW124, 500 ms
   "2920RS001A01T05.FP_PARAM.AlarmDelay_L1_Acc" : Int AT %DB5056.DBW126, 500 ms
   "2920RS001A01T05.FP_PARAM.AlarmDelay_L2_Pre" : Int AT %DB5056.DBW128, 500 ms
   "2920RS001A01T05.FP_PARAM.AlarmDelay_L2_Acc" : Int AT %DB5056.DBW130, 500 ms
   "2920RS001A01T05.FP_PARAM.AlarmDelay_L3_Pre" : Int AT %DB5056.DBW132, 500 ms
   "2920RS001A01T05.FP_PARAM.AlarmDelay_L3_Acc" : Int AT %DB5056.DBW134, 500 ms
   "2920RS001A01T05.FP_PARAM.OpenLoopDelay_Pre" : Int AT %DB5056.DBW136, 500 ms
   "2920RS001A01T05.FP_PARAM.OpenLoopDelay_Acc" : Int AT %DB5056.DBW138, 500 ms
   "2920RS001A01T05.FP_PARAM.OverRangeDelay_Pre" : Int AT %DB5056.DBW140, 500 ms
   "2920RS001A01T05.FP_PARAM.OverRangeDelay_Acc" : Int AT %DB5056.DBW142, 500 ms
   "2920RS001A01T05.FP_PARAM.AuxLimit_H2_Value" : Real AT %DB5056.DBD144, 500 ms
   "2920RS001A01T05.FP_PARAM.AuxLimit_H1_Value" : Real AT %DB5056.DBD148, 500 ms
   "2920RS001A01T05.FP_PARAM.AuxLimit_L2_Value" : Real AT %DB5056.DBD152, 500 ms
   "2920RS001A01T05.FP_PARAM.AuxLimit_L1_Value" : Real AT %DB5056.DBD156, 500 ms
   "2920RS001A01T05.Unit" : TextRef, internal   // Еденицы измерения При експорте из ECS через скрипт заполняется автоматически, если теги копируются в ручную то требуется задатать свойство Text
   "2920RS001A01T05.Decimals" : TextRef, internal   // Формат отображения При експорте из ECS через скрипт, заполняется автоматически. Если теги копируются в ручную то требуется задатать свойство Text s999999.9
   "2920RS001A01T05.FP_EN.Square" : Bool AT %DB5056.DBX46.0, 500 ms
   "2920RS001A01T05.FP_EN.SquareRoot" : Bool AT %DB5056.DBX46.1, 500 ms
   "2920RS001A01T05.FP_EN.ParentSupress" : Bool AT %DB5056.DBX46.2, 500 ms
   "2920RS001A01T05.FP_EN.ParentSupressUnit" : Bool AT %DB5056.DBX46.3, 500 ms
   "2920RS001A01T05.FP_EN.Force" : Bool AT %DB5056.DBX46.4, 500 ms
   "2920RS001A01T05.FP_EN.Damping" : Bool AT %DB5056.DBX46.5, 500 ms
   "2920RS001A01T05.FP_EN.Gradient_Pos" : Bool AT %DB5056.DBX46.6, 500 ms
   "2920RS001A01T05.FP_EN.Gradient_Neg" : Bool AT %DB5056.DBX46.7, 500 ms
   "2920RS001A01T05.FP_EN.Hysteresis" : Bool AT %DB5056.DBX47.0, 500 ms
   "2920RS001A01T05.FP_EN.Alarm_H3" : Bool AT %DB5056.DBX47.1, 500 ms
   "2920RS001A01T05.FP_EN.Alarm_H2" : Bool AT %DB5056.DBX47.2, 500 ms
   "2920RS001A01T05.FP_EN.Alarm_H1" : Bool AT %DB5056.DBX47.3, 500 ms
   "2920RS001A01T05.FP_EN.Alarm_L1" : Bool AT %DB5056.DBX47.4, 500 ms
   "2920RS001A01T05.FP_EN.Alarm_L2" : Bool AT %DB5056.DBX47.5, 500 ms
   "2920RS001A01T05.FP_EN.Alarm_L3" : Bool AT %DB5056.DBX47.6, 500 ms
   "2920RS001A01T05.FP_EN.AlarmDelay_H3" : Bool AT %DB5056.DBX47.7, 500 ms
   "2920RS001A01T05.FP_EN.AlarmDelay_H2" : Bool AT %DB5056.DBX48.0, 500 ms
   "2920RS001A01T05.FP_EN.AlarmDelay_H1" : Bool AT %DB5056.DBX48.1, 500 ms
   "2920RS001A01T05.FP_EN.AlarmDelay_L1" : Bool AT %DB5056.DBX48.2, 500 ms
   "2920RS001A01T05.FP_EN.AlarmDelay_L2" : Bool AT %DB5056.DBX48.3, 500 ms
   "2920RS001A01T05.FP_EN.AlarmDelay_L3" : Bool AT %DB5056.DBX48.4, 500 ms
   "2920RS001A01T05.FP_EN.ROC_Warn" : Bool AT %DB5056.DBX48.5, 500 ms
   "2920RS001A01T05.FP_EN.U_Range_Warn" : Bool AT %DB5056.DBX48.6, 500 ms
   "2920RS001A01T05.FP_EN.O_Range_Warn" : Bool AT %DB5056.DBX48.7, 500 ms
   "2920RS001A01T05.trend_tag_name" : TextRef, internal   // Еденицы измерения При експорте из ECS через скрипт - заполняется автоматически, если теги копируются в ручную то требуется задатать свойство Text - имя тега для тренда
   "2920RS001A01T05.DQ.AL_H3" : Bool AT %DB5056.DBX16.0, 500 ms
   "2920RS001A01T05.DQ.AL_H2" : Bool AT %DB5056.DBX16.1, 500 ms
   "2920RS001A01T05.DQ.AL_H1" : Bool AT %DB5056.DBX16.2, 500 ms
   "2920RS001A01T05.DQ.AL_L1" : Bool AT %DB5056.DBX16.3, 500 ms
   "2920RS001A01T05.DQ.AL_L2" : Bool AT %DB5056.DBX16.4, 500 ms
   "2920RS001A01T05.DQ.AL_L3" : Bool AT %DB5056.DBX16.5, 500 ms
   "2920RS001A01T05.DQ.SIG_OK" : Bool AT %DB5056.DBX16.6, 500 ms
   "2920RS001A01T05.DQ.LIM_H2" : Bool AT %DB5056.DBX16.7, 500 ms
   "2920RS001A01T05.DQ.LIM_H1" : Bool AT %DB5056.DBX17.0, 500 ms
   "2920RS001A01T05.DQ.LIM_L1" : Bool AT %DB5056.DBX17.1, 500 ms
   "2920RS001A01T05.DQ.LIM_L2" : Bool AT %DB5056.DBX17.2, 500 ms
   "2920RS001A01T05.DQ.GR_P" : Bool AT %DB5056.DBX17.3, 500 ms
   "2920RS001A01T05.DQ.GR_N" : Bool AT %DB5056.DBX17.4, 500 ms
   "2920RS001A01T05.I.IN" : Real AT %DB5056.DBD2, 500 ms
   "2920RS001A01T05.I.SIG_TYPE" : Int AT %DB5056.DBW0, 500 ms
   "2920RS001A01T05.I.FI_BUS" : Byte AT %DB5056.DBB6, 500 ms
   "2920RS001A01T05.DI.U_RANGE" : Bool AT %DB5056.DBX7.0, 500 ms
   "2920RS001A01T05.DI.O_RANGE" : Bool AT %DB5056.DBX7.1, 500 ms
   "2920RS001A01T05.DI.SIG_FAULT" : Bool AT %DB5056.DBX7.2, 500 ms
   "2920RS001A01T05.DI.EnConfig" : Bool AT %DB5056.DBX7.3, 500 ms
   "2920RS001A01T05.DI.AEN" : Bool AT %DB5056.DBX7.4, 500 ms
   "2920RS001A01T05.DI.AL_SUPR" : Bool AT %DB5056.DBX7.5, 500 ms
   "2920RS001A01T05.Q.PV_NORM" : Real AT %DB5056.DBD8, 500 ms
   "2920RS001A01T05.Q.PV_SCAL" : Real AT %DB5056.DBD12, 500 ms
   "2920RS001A01T05.ParentInfo" : TextRef, internal   // Имя родителя для попап окна, вкладка инфо. При експорте из ECS через скрипт заполняется автоматически, если теги копируются в ручную то требуется в ручную задатать свойство Start Value

HMI tags "2920RS001A01T06"
   "2920RS001A01T06.MSW" : 52809b66-421d-457f-8884-6f7a49d4e247 AT %DB5057.DBX18.0, 500 ms
   "2920RS001A01T06.DefaultText" : TextRef, internal   // Заголовок POPUP окна. При експорте из ECS через скрипт заполняется автоматически, если теги копируются в ручную то требуется в ручную задатать свойство Start Value
   "2920RS001A01T06.BlockInfo" : Array [0..2] of Int AT %DB5057.DBX38.0, 500 ms
   "2920RS001A01T06.StatusWork" : Int AT %DB5057.DBW242, 500 ms
   "2920RS001A01T06.FP_PARAM.DampingTime" : Int AT %DB5057.DBW50, 500 ms
   "2920RS001A01T06.FP_PARAM.Force_Value" : Real AT %DB5057.DBD52, 500 ms
   "2920RS001A01T06.FP_PARAM.Scale_Min" : Real AT %DB5057.DBD56, 500 ms
   "2920RS001A01T06.FP_PARAM.Scale_Max" : Real AT %DB5057.DBD60, 500 ms
   "2920RS001A01T06.FP_PARAM.Gradient" : Real AT %DB5057.DBD64, 500 ms
   "2920RS001A01T06.FP_PARAM.Grad_Pos" : Real AT %DB5057.DBD68, 500 ms
   "2920RS001A01T06.FP_PARAM.Grad_Neg" : Real AT %DB5057.DBD72, 500 ms
   "2920RS001A01T06.FP_PARAM.Grad_X" : Real AT %DB5057.DBD76, 500 ms
   "2920RS001A01T06.FP_PARAM.Gradient_Time_Pre" : Int AT %DB5057.DBW80, 500 ms
   "2920RS001A01T06.FP_PARAM.Gradient_Time_ACC" : Int AT %DB5057.DBW82, 500 ms
   "2920RS001A01T06.FP_PARAM.Alarm_Hyst" : Real AT %DB5057.DBD84, 500 ms
   "2920RS001A01T06.FP_PARAM.AlarmLimit_H3" : Real AT %DB5057.DBD88, 500 ms
   "2920RS001A01T06.FP_PARAM.AlarmLimit_H2" : Real AT %DB5057.DBD92, 500 ms
   "2920RS001A01T06.FP_PARAM.AlarmLimit_H1" : Real AT %DB5057.DBD96, 500 ms
   "2920RS001A01T06.FP_PARAM.AlarmLimit_L1" : Real AT %DB5057.DBD100, 500 ms
   "2920RS001A01T06.FP_PARAM.AlarmLimit_L2" : Real AT %DB5057.DBD104, 500 ms
   "2920RS001A01T06.FP_PARAM.AlarmLimit_L3" : Real AT %DB5057.DBD108, 500 ms
   "2920RS001A01T06.FP_PARAM.AlarmDelay_H3_Pre" : Int AT %DB5057.DBW112, 500 ms
   "2920RS001A01T06.FP_PARAM.AlarmDelay_H3_Acc" : Int AT %DB5057.DBW114, 500 ms
   "2920RS001A01T06.FP_PARAM.AlarmDelay_H2_Pre" : Int AT %DB5057.DBW116, 500 ms
   "2920RS001A01T06.FP_PARAM.AlarmDelay_H2_Acc" : Int AT %DB5057.DBW118, 500 ms
   "2920RS001A01T06.FP_PARAM.AlarmDelay_H1_Pre" : Int AT %DB5057.DBW120, 500 ms
   "2920RS001A01T06.FP_PARAM.AlarmDelay_H1_Acc" : Int AT %DB5057.DBW122, 500 ms
   "2920RS001A01T06.FP_PARAM.AlarmDelay_L1_Pre" : Int AT %DB5057.DBW124, 500 ms
   "2920RS001A01T06.FP_PARAM.AlarmDelay_L1_Acc" : Int AT %DB5057.DBW126, 500 ms
   "2920RS001A01T06.FP_PARAM.AlarmDelay_L2_Pre" : Int AT %DB5057.DBW128, 500 ms
   "2920RS001A01T06.FP_PARAM.AlarmDelay_L2_Acc" : Int AT %DB5057.DBW130, 500 ms
   "2920RS001A01T06.FP_PARAM.AlarmDelay_L3_Pre" : Int AT %DB5057.DBW132, 500 ms
   "2920RS001A01T06.FP_PARAM.AlarmDelay_L3_Acc" : Int AT %DB5057.DBW134, 500 ms
   "2920RS001A01T06.FP_PARAM.OpenLoopDelay_Pre" : Int AT %DB5057.DBW136, 500 ms
   "2920RS001A01T06.FP_PARAM.OpenLoopDelay_Acc" : Int AT %DB5057.DBW138, 500 ms
   "2920RS001A01T06.FP_PARAM.OverRangeDelay_Pre" : Int AT %DB5057.DBW140, 500 ms
   "2920RS001A01T06.FP_PARAM.OverRangeDelay_Acc" : Int AT %DB5057.DBW142, 500 ms
   "2920RS001A01T06.FP_PARAM.AuxLimit_H2_Value" : Real AT %DB5057.DBD144, 500 ms
   "2920RS001A01T06.FP_PARAM.AuxLimit_H1_Value" : Real AT %DB5057.DBD148, 500 ms
   "2920RS001A01T06.FP_PARAM.AuxLimit_L2_Value" : Real AT %DB5057.DBD152, 500 ms
   "2920RS001A01T06.FP_PARAM.AuxLimit_L1_Value" : Real AT %DB5057.DBD156, 500 ms
   "2920RS001A01T06.Unit" : TextRef, internal   // Еденицы измерения При експорте из ECS через скрипт заполняется автоматически, если теги копируются в ручную то требуется задатать свойство Text
   "2920RS001A01T06.Decimals" : TextRef, internal   // Формат отображения При експорте из ECS через скрипт, заполняется автоматически. Если теги копируются в ручную то требуется задатать свойство Text s999999.9
   "2920RS001A01T06.FP_EN.Square" : Bool AT %DB5057.DBX46.0, 500 ms
   "2920RS001A01T06.FP_EN.SquareRoot" : Bool AT %DB5057.DBX46.1, 500 ms
   "2920RS001A01T06.FP_EN.ParentSupress" : Bool AT %DB5057.DBX46.2, 500 ms
   "2920RS001A01T06.FP_EN.ParentSupressUnit" : Bool AT %DB5057.DBX46.3, 500 ms
   "2920RS001A01T06.FP_EN.Force" : Bool AT %DB5057.DBX46.4, 500 ms
   "2920RS001A01T06.FP_EN.Damping" : Bool AT %DB5057.DBX46.5, 500 ms
   "2920RS001A01T06.FP_EN.Gradient_Pos" : Bool AT %DB5057.DBX46.6, 500 ms
   "2920RS001A01T06.FP_EN.Gradient_Neg" : Bool AT %DB5057.DBX46.7, 500 ms
   "2920RS001A01T06.FP_EN.Hysteresis" : Bool AT %DB5057.DBX47.0, 500 ms
   "2920RS001A01T06.FP_EN.Alarm_H3" : Bool AT %DB5057.DBX47.1, 500 ms
   "2920RS001A01T06.FP_EN.Alarm_H2" : Bool AT %DB5057.DBX47.2, 500 ms
   "2920RS001A01T06.FP_EN.Alarm_H1" : Bool AT %DB5057.DBX47.3, 500 ms
   "2920RS001A01T06.FP_EN.Alarm_L1" : Bool AT %DB5057.DBX47.4, 500 ms
   "2920RS001A01T06.FP_EN.Alarm_L2" : Bool AT %DB5057.DBX47.5, 500 ms
   "2920RS001A01T06.FP_EN.Alarm_L3" : Bool AT %DB5057.DBX47.6, 500 ms
   "2920RS001A01T06.FP_EN.AlarmDelay_H3" : Bool AT %DB5057.DBX47.7, 500 ms
   "2920RS001A01T06.FP_EN.AlarmDelay_H2" : Bool AT %DB5057.DBX48.0, 500 ms
   "2920RS001A01T06.FP_EN.AlarmDelay_H1" : Bool AT %DB5057.DBX48.1, 500 ms
   "2920RS001A01T06.FP_EN.AlarmDelay_L1" : Bool AT %DB5057.DBX48.2, 500 ms
   "2920RS001A01T06.FP_EN.AlarmDelay_L2" : Bool AT %DB5057.DBX48.3, 500 ms
   "2920RS001A01T06.FP_EN.AlarmDelay_L3" : Bool AT %DB5057.DBX48.4, 500 ms
   "2920RS001A01T06.FP_EN.ROC_Warn" : Bool AT %DB5057.DBX48.5, 500 ms
   "2920RS001A01T06.FP_EN.U_Range_Warn" : Bool AT %DB5057.DBX48.6, 500 ms
   "2920RS001A01T06.FP_EN.O_Range_Warn" : Bool AT %DB5057.DBX48.7, 500 ms
   "2920RS001A01T06.trend_tag_name" : TextRef, internal   // Еденицы измерения При експорте из ECS через скрипт - заполняется автоматически, если теги копируются в ручную то требуется задатать свойство Text - имя тега для тренда
   "2920RS001A01T06.DQ.AL_H3" : Bool AT %DB5057.DBX16.0, 500 ms
   "2920RS001A01T06.DQ.AL_H2" : Bool AT %DB5057.DBX16.1, 500 ms
   "2920RS001A01T06.DQ.AL_H1" : Bool AT %DB5057.DBX16.2, 500 ms
   "2920RS001A01T06.DQ.AL_L1" : Bool AT %DB5057.DBX16.3, 500 ms
   "2920RS001A01T06.DQ.AL_L2" : Bool AT %DB5057.DBX16.4, 500 ms
   "2920RS001A01T06.DQ.AL_L3" : Bool AT %DB5057.DBX16.5, 500 ms
   "2920RS001A01T06.DQ.SIG_OK" : Bool AT %DB5057.DBX16.6, 500 ms
   "2920RS001A01T06.DQ.LIM_H2" : Bool AT %DB5057.DBX16.7, 500 ms
   "2920RS001A01T06.DQ.LIM_H1" : Bool AT %DB5057.DBX17.0, 500 ms
   "2920RS001A01T06.DQ.LIM_L1" : Bool AT %DB5057.DBX17.1, 500 ms
   "2920RS001A01T06.DQ.LIM_L2" : Bool AT %DB5057.DBX17.2, 500 ms
   "2920RS001A01T06.DQ.GR_P" : Bool AT %DB5057.DBX17.3, 500 ms
   "2920RS001A01T06.DQ.GR_N" : Bool AT %DB5057.DBX17.4, 500 ms
   "2920RS001A01T06.I.IN" : Real AT %DB5057.DBD2, 500 ms
   "2920RS001A01T06.I.SIG_TYPE" : Int AT %DB5057.DBW0, 500 ms
   "2920RS001A01T06.I.FI_BUS" : Byte AT %DB5057.DBB6, 500 ms
   "2920RS001A01T06.DI.U_RANGE" : Bool AT %DB5057.DBX7.0, 500 ms
   "2920RS001A01T06.DI.O_RANGE" : Bool AT %DB5057.DBX7.1, 500 ms
   "2920RS001A01T06.DI.SIG_FAULT" : Bool AT %DB5057.DBX7.2, 500 ms
   "2920RS001A01T06.DI.EnConfig" : Bool AT %DB5057.DBX7.3, 500 ms
   "2920RS001A01T06.DI.AEN" : Bool AT %DB5057.DBX7.4, 500 ms
   "2920RS001A01T06.DI.AL_SUPR" : Bool AT %DB5057.DBX7.5, 500 ms
   "2920RS001A01T06.Q.PV_NORM" : Real AT %DB5057.DBD8, 500 ms
   "2920RS001A01T06.Q.PV_SCAL" : Real AT %DB5057.DBD12, 500 ms
   "2920RS001A01T06.ParentInfo" : TextRef, internal   // Имя родителя для попап окна, вкладка инфо. При експорте из ECS через скрипт заполняется автоматически, если теги копируются в ручную то требуется в ручную задатать свойство Start Value

HMI tags "2925RS001A01F01"
   "2925RS001A01F01.MSW" : 52809b66-421d-457f-8884-6f7a49d4e247 AT %DB5058.DBX18.0, 500 ms
   "2925RS001A01F01.DefaultText" : TextRef, internal   // Заголовок POPUP окна. При експорте из ECS через скрипт заполняется автоматически, если теги копируются в ручную то требуется в ручную задатать свойство Start Value
   "2925RS001A01F01.BlockInfo" : Array [0..2] of Int AT %DB5058.DBX38.0, 500 ms
   "2925RS001A01F01.StatusWork" : Int AT %DB5058.DBW242, 500 ms
   "2925RS001A01F01.FP_PARAM.DampingTime" : Int AT %DB5058.DBW50, 500 ms
   "2925RS001A01F01.FP_PARAM.Force_Value" : Real AT %DB5058.DBD52, 500 ms
   "2925RS001A01F01.FP_PARAM.Scale_Min" : Real AT %DB5058.DBD56, 500 ms
   "2925RS001A01F01.FP_PARAM.Scale_Max" : Real AT %DB5058.DBD60, 500 ms
   "2925RS001A01F01.FP_PARAM.Gradient" : Real AT %DB5058.DBD64, 500 ms
   "2925RS001A01F01.FP_PARAM.Grad_Pos" : Real AT %DB5058.DBD68, 500 ms
   "2925RS001A01F01.FP_PARAM.Grad_Neg" : Real AT %DB5058.DBD72, 500 ms
   "2925RS001A01F01.FP_PARAM.Grad_X" : Real AT %DB5058.DBD76, 500 ms
   "2925RS001A01F01.FP_PARAM.Gradient_Time_Pre" : Int AT %DB5058.DBW80, 500 ms
   "2925RS001A01F01.FP_PARAM.Gradient_Time_ACC" : Int AT %DB5058.DBW82, 500 ms
   "2925RS001A01F01.FP_PARAM.Alarm_Hyst" : Real AT %DB5058.DBD84, 500 ms
   "2925RS001A01F01.FP_PARAM.AlarmLimit_H3" : Real AT %DB5058.DBD88, 500 ms
   "2925RS001A01F01.FP_PARAM.AlarmLimit_H2" : Real AT %DB5058.DBD92, 500 ms
   "2925RS001A01F01.FP_PARAM.AlarmLimit_H1" : Real AT %DB5058.DBD96, 500 ms
   "2925RS001A01F01.FP_PARAM.AlarmLimit_L1" : Real AT %DB5058.DBD100, 500 ms
   "2925RS001A01F01.FP_PARAM.AlarmLimit_L2" : Real AT %DB5058.DBD104, 500 ms
   "2925RS001A01F01.FP_PARAM.AlarmLimit_L3" : Real AT %DB5058.DBD108, 500 ms
   "2925RS001A01F01.FP_PARAM.AlarmDelay_H3_Pre" : Int AT %DB5058.DBW112, 500 ms
   "2925RS001A01F01.FP_PARAM.AlarmDelay_H3_Acc" : Int AT %DB5058.DBW114, 500 ms
   "2925RS001A01F01.FP_PARAM.AlarmDelay_H2_Pre" : Int AT %DB5058.DBW116, 500 ms
   "2925RS001A01F01.FP_PARAM.AlarmDelay_H2_Acc" : Int AT %DB5058.DBW118, 500 ms
   "2925RS001A01F01.FP_PARAM.AlarmDelay_H1_Pre" : Int AT %DB5058.DBW120, 500 ms
   "2925RS001A01F01.FP_PARAM.AlarmDelay_H1_Acc" : Int AT %DB5058.DBW122, 500 ms
   "2925RS001A01F01.FP_PARAM.AlarmDelay_L1_Pre" : Int AT %DB5058.DBW124, 500 ms
   "2925RS001A01F01.FP_PARAM.AlarmDelay_L1_Acc" : Int AT %DB5058.DBW126, 500 ms
   "2925RS001A01F01.FP_PARAM.AlarmDelay_L2_Pre" : Int AT %DB5058.DBW128, 500 ms
   "2925RS001A01F01.FP_PARAM.AlarmDelay_L2_Acc" : Int AT %DB5058.DBW130, 500 ms
   "2925RS001A01F01.FP_PARAM.AlarmDelay_L3_Pre" : Int AT %DB5058.DBW132, 500 ms
   "2925RS001A01F01.FP_PARAM.AlarmDelay_L3_Acc" : Int AT %DB5058.DBW134, 500 ms
   "2925RS001A01F01.FP_PARAM.OpenLoopDelay_Pre" : Int AT %DB5058.DBW136, 500 ms
   "2925RS001A01F01.FP_PARAM.OpenLoopDelay_Acc" : Int AT %DB5058.DBW138, 500 ms
   "2925RS001A01F01.FP_PARAM.OverRangeDelay_Pre" : Int AT %DB5058.DBW140, 500 ms
   "2925RS001A01F01.FP_PARAM.OverRangeDelay_Acc" : Int AT %DB5058.DBW142, 500 ms
   "2925RS001A01F01.FP_PARAM.AuxLimit_H2_Value" : Real AT %DB5058.DBD144, 500 ms
   "2925RS001A01F01.FP_PARAM.AuxLimit_H1_Value" : Real AT %DB5058.DBD148, 500 ms
   "2925RS001A01F01.FP_PARAM.AuxLimit_L2_Value" : Real AT %DB5058.DBD152, 500 ms
   "2925RS001A01F01.FP_PARAM.AuxLimit_L1_Value" : Real AT %DB5058.DBD156, 500 ms
   "2925RS001A01F01.Unit" : TextRef, internal   // Еденицы измерения При експорте из ECS через скрипт заполняется автоматически, если теги копируются в ручную то требуется задатать свойство Text
   "2925RS001A01F01.Decimals" : TextRef, internal   // Формат отображения При експорте из ECS через скрипт, заполняется автоматически. Если теги копируются в ручную то требуется задатать свойство Text s999999.9
   "2925RS001A01F01.FP_EN.Square" : Bool AT %DB5058.DBX46.0, 500 ms
   "2925RS001A01F01.FP_EN.SquareRoot" : Bool AT %DB5058.DBX46.1, 500 ms
   "2925RS001A01F01.FP_EN.ParentSupress" : Bool AT %DB5058.DBX46.2, 500 ms
   "2925RS001A01F01.FP_EN.ParentSupressUnit" : Bool AT %DB5058.DBX46.3, 500 ms
   "2925RS001A01F01.FP_EN.Force" : Bool AT %DB5058.DBX46.4, 500 ms
   "2925RS001A01F01.FP_EN.Damping" : Bool AT %DB5058.DBX46.5, 500 ms
   "2925RS001A01F01.FP_EN.Gradient_Pos" : Bool AT %DB5058.DBX46.6, 500 ms
   "2925RS001A01F01.FP_EN.Gradient_Neg" : Bool AT %DB5058.DBX46.7, 500 ms
   "2925RS001A01F01.FP_EN.Hysteresis" : Bool AT %DB5058.DBX47.0, 500 ms
   "2925RS001A01F01.FP_EN.Alarm_H3" : Bool AT %DB5058.DBX47.1, 500 ms
   "2925RS001A01F01.FP_EN.Alarm_H2" : Bool AT %DB5058.DBX47.2, 500 ms
   "2925RS001A01F01.FP_EN.Alarm_H1" : Bool AT %DB5058.DBX47.3, 500 ms
   "2925RS001A01F01.FP_EN.Alarm_L1" : Bool AT %DB5058.DBX47.4, 500 ms
   "2925RS001A01F01.FP_EN.Alarm_L2" : Bool AT %DB5058.DBX47.5, 500 ms
   "2925RS001A01F01.FP_EN.Alarm_L3" : Bool AT %DB5058.DBX47.6, 500 ms
   "2925RS001A01F01.FP_EN.AlarmDelay_H3" : Bool AT %DB5058.DBX47.7, 500 ms
   "2925RS001A01F01.FP_EN.AlarmDelay_H2" : Bool AT %DB5058.DBX48.0, 500 ms
   "2925RS001A01F01.FP_EN.AlarmDelay_H1" : Bool AT %DB5058.DBX48.1, 500 ms
   "2925RS001A01F01.FP_EN.AlarmDelay_L1" : Bool AT %DB5058.DBX48.2, 500 ms
   "2925RS001A01F01.FP_EN.AlarmDelay_L2" : Bool AT %DB5058.DBX48.3, 500 ms
   "2925RS001A01F01.FP_EN.AlarmDelay_L3" : Bool AT %DB5058.DBX48.4, 500 ms
   "2925RS001A01F01.FP_EN.ROC_Warn" : Bool AT %DB5058.DBX48.5, 500 ms
   "2925RS001A01F01.FP_EN.U_Range_Warn" : Bool AT %DB5058.DBX48.6, 500 ms
   "2925RS001A01F01.FP_EN.O_Range_Warn" : Bool AT %DB5058.DBX48.7, 500 ms
   "2925RS001A01F01.trend_tag_name" : TextRef, internal   // Еденицы измерения При експорте из ECS через скрипт - заполняется автоматически, если теги копируются в ручную то требуется задатать свойство Text - имя тега для тренда
   "2925RS001A01F01.DQ.AL_H3" : Bool AT %DB5058.DBX16.0, 500 ms
   "2925RS001A01F01.DQ.AL_H2" : Bool AT %DB5058.DBX16.1, 500 ms
   "2925RS001A01F01.DQ.AL_H1" : Bool AT %DB5058.DBX16.2, 500 ms
   "2925RS001A01F01.DQ.AL_L1" : Bool AT %DB5058.DBX16.3, 500 ms
   "2925RS001A01F01.DQ.AL_L2" : Bool AT %DB5058.DBX16.4, 500 ms
   "2925RS001A01F01.DQ.AL_L3" : Bool AT %DB5058.DBX16.5, 500 ms
   "2925RS001A01F01.DQ.SIG_OK" : Bool AT %DB5058.DBX16.6, 500 ms
   "2925RS001A01F01.DQ.LIM_H2" : Bool AT %DB5058.DBX16.7, 500 ms
   "2925RS001A01F01.DQ.LIM_H1" : Bool AT %DB5058.DBX17.0, 500 ms
   "2925RS001A01F01.DQ.LIM_L1" : Bool AT %DB5058.DBX17.1, 500 ms
   "2925RS001A01F01.DQ.LIM_L2" : Bool AT %DB5058.DBX17.2, 500 ms
   "2925RS001A01F01.DQ.GR_P" : Bool AT %DB5058.DBX17.3, 500 ms
   "2925RS001A01F01.DQ.GR_N" : Bool AT %DB5058.DBX17.4, 500 ms
   "2925RS001A01F01.I.IN" : Real AT %DB5058.DBD2, 500 ms
   "2925RS001A01F01.I.SIG_TYPE" : Int AT %DB5058.DBW0, 500 ms
   "2925RS001A01F01.I.FI_BUS" : Byte AT %DB5058.DBB6, 500 ms
   "2925RS001A01F01.DI.U_RANGE" : Bool AT %DB5058.DBX7.0, 500 ms
   "2925RS001A01F01.DI.O_RANGE" : Bool AT %DB5058.DBX7.1, 500 ms
   "2925RS001A01F01.DI.SIG_FAULT" : Bool AT %DB5058.DBX7.2, 500 ms
   "2925RS001A01F01.DI.EnConfig" : Bool AT %DB5058.DBX7.3, 500 ms
   "2925RS001A01F01.DI.AEN" : Bool AT %DB5058.DBX7.4, 500 ms
   "2925RS001A01F01.DI.AL_SUPR" : Bool AT %DB5058.DBX7.5, 500 ms
   "2925RS001A01F01.Q.PV_NORM" : Real AT %DB5058.DBD8, 500 ms
   "2925RS001A01F01.Q.PV_SCAL" : Real AT %DB5058.DBD12, 500 ms
   "2925RS001A01F01.ParentInfo" : TextRef, internal   // Имя родителя для попап окна, вкладка инфо. При експорте из ECS через скрипт заполняется автоматически, если теги копируются в ручную то требуется в ручную задатать свойство Start Value

HMI tags "2925RS001A01F02"
   "2925RS001A01F02.MSW" : 52809b66-421d-457f-8884-6f7a49d4e247 AT %DB5059.DBX18.0, 500 ms
   "2925RS001A01F02.DefaultText" : TextRef, internal   // Заголовок POPUP окна. При експорте из ECS через скрипт заполняется автоматически, если теги копируются в ручную то требуется в ручную задатать свойство Start Value
   "2925RS001A01F02.BlockInfo" : Array [0..2] of Int AT %DB5059.DBX38.0, 500 ms
   "2925RS001A01F02.StatusWork" : Int AT %DB5059.DBW242, 500 ms
   "2925RS001A01F02.FP_PARAM.DampingTime" : Int AT %DB5059.DBW50, 500 ms
   "2925RS001A01F02.FP_PARAM.Force_Value" : Real AT %DB5059.DBD52, 500 ms
   "2925RS001A01F02.FP_PARAM.Scale_Min" : Real AT %DB5059.DBD56, 500 ms
   "2925RS001A01F02.FP_PARAM.Scale_Max" : Real AT %DB5059.DBD60, 500 ms
   "2925RS001A01F02.FP_PARAM.Gradient" : Real AT %DB5059.DBD64, 500 ms
   "2925RS001A01F02.FP_PARAM.Grad_Pos" : Real AT %DB5059.DBD68, 500 ms
   "2925RS001A01F02.FP_PARAM.Grad_Neg" : Real AT %DB5059.DBD72, 500 ms
   "2925RS001A01F02.FP_PARAM.Grad_X" : Real AT %DB5059.DBD76, 500 ms
   "2925RS001A01F02.FP_PARAM.Gradient_Time_Pre" : Int AT %DB5059.DBW80, 500 ms
   "2925RS001A01F02.FP_PARAM.Gradient_Time_ACC" : Int AT %DB5059.DBW82, 500 ms
   "2925RS001A01F02.FP_PARAM.Alarm_Hyst" : Real AT %DB5059.DBD84, 500 ms
   "2925RS001A01F02.FP_PARAM.AlarmLimit_H3" : Real AT %DB5059.DBD88, 500 ms
   "2925RS001A01F02.FP_PARAM.AlarmLimit_H2" : Real AT %DB5059.DBD92, 500 ms
   "2925RS001A01F02.FP_PARAM.AlarmLimit_H1" : Real AT %DB5059.DBD96, 500 ms
   "2925RS001A01F02.FP_PARAM.AlarmLimit_L1" : Real AT %DB5059.DBD100, 500 ms
   "2925RS001A01F02.FP_PARAM.AlarmLimit_L2" : Real AT %DB5059.DBD104, 500 ms
   "2925RS001A01F02.FP_PARAM.AlarmLimit_L3" : Real AT %DB5059.DBD108, 500 ms
   "2925RS001A01F02.FP_PARAM.AlarmDelay_H3_Pre" : Int AT %DB5059.DBW112, 500 ms
   "2925RS001A01F02.FP_PARAM.AlarmDelay_H3_Acc" : Int AT %DB5059.DBW114, 500 ms
   "2925RS001A01F02.FP_PARAM.AlarmDelay_H2_Pre" : Int AT %DB5059.DBW116, 500 ms
   "2925RS001A01F02.FP_PARAM.AlarmDelay_H2_Acc" : Int AT %DB5059.DBW118, 500 ms
   "2925RS001A01F02.FP_PARAM.AlarmDelay_H1_Pre" : Int AT %DB5059.DBW120, 500 ms
   "2925RS001A01F02.FP_PARAM.AlarmDelay_H1_Acc" : Int AT %DB5059.DBW122, 500 ms
   "2925RS001A01F02.FP_PARAM.AlarmDelay_L1_Pre" : Int AT %DB5059.DBW124, 500 ms
   "2925RS001A01F02.FP_PARAM.AlarmDelay_L1_Acc" : Int AT %DB5059.DBW126, 500 ms
   "2925RS001A01F02.FP_PARAM.AlarmDelay_L2_Pre" : Int AT %DB5059.DBW128, 500 ms
   "2925RS001A01F02.FP_PARAM.AlarmDelay_L2_Acc" : Int AT %DB5059.DBW130, 500 ms
   "2925RS001A01F02.FP_PARAM.AlarmDelay_L3_Pre" : Int AT %DB5059.DBW132, 500 ms
   "2925RS001A01F02.FP_PARAM.AlarmDelay_L3_Acc" : Int AT %DB5059.DBW134, 500 ms
   "2925RS001A01F02.FP_PARAM.OpenLoopDelay_Pre" : Int AT %DB5059.DBW136, 500 ms
   "2925RS001A01F02.FP_PARAM.OpenLoopDelay_Acc" : Int AT %DB5059.DBW138, 500 ms
   "2925RS001A01F02.FP_PARAM.OverRangeDelay_Pre" : Int AT %DB5059.DBW140, 500 ms
   "2925RS001A01F02.FP_PARAM.OverRangeDelay_Acc" : Int AT %DB5059.DBW142, 500 ms
   "2925RS001A01F02.FP_PARAM.AuxLimit_H2_Value" : Real AT %DB5059.DBD144, 500 ms
   "2925RS001A01F02.FP_PARAM.AuxLimit_H1_Value" : Real AT %DB5059.DBD148, 500 ms
   "2925RS001A01F02.FP_PARAM.AuxLimit_L2_Value" : Real AT %DB5059.DBD152, 500 ms
   "2925RS001A01F02.FP_PARAM.AuxLimit_L1_Value" : Real AT %DB5059.DBD156, 500 ms
   "2925RS001A01F02.Unit" : TextRef, internal   // Еденицы измерения При експорте из ECS через скрипт заполняется автоматически, если теги копируются в ручную то требуется задатать свойство Text
   "2925RS001A01F02.Decimals" : TextRef, internal   // Формат отображения При експорте из ECS через скрипт, заполняется автоматически. Если теги копируются в ручную то требуется задатать свойство Text s999999.9
   "2925RS001A01F02.FP_EN.Square" : Bool AT %DB5059.DBX46.0, 500 ms
   "2925RS001A01F02.FP_EN.SquareRoot" : Bool AT %DB5059.DBX46.1, 500 ms
   "2925RS001A01F02.FP_EN.ParentSupress" : Bool AT %DB5059.DBX46.2, 500 ms
   "2925RS001A01F02.FP_EN.ParentSupressUnit" : Bool AT %DB5059.DBX46.3, 500 ms
   "2925RS001A01F02.FP_EN.Force" : Bool AT %DB5059.DBX46.4, 500 ms
   "2925RS001A01F02.FP_EN.Damping" : Bool AT %DB5059.DBX46.5, 500 ms
   "2925RS001A01F02.FP_EN.Gradient_Pos" : Bool AT %DB5059.DBX46.6, 500 ms
   "2925RS001A01F02.FP_EN.Gradient_Neg" : Bool AT %DB5059.DBX46.7, 500 ms
   "2925RS001A01F02.FP_EN.Hysteresis" : Bool AT %DB5059.DBX47.0, 500 ms
   "2925RS001A01F02.FP_EN.Alarm_H3" : Bool AT %DB5059.DBX47.1, 500 ms
   "2925RS001A01F02.FP_EN.Alarm_H2" : Bool AT %DB5059.DBX47.2, 500 ms
   "2925RS001A01F02.FP_EN.Alarm_H1" : Bool AT %DB5059.DBX47.3, 500 ms
   "2925RS001A01F02.FP_EN.Alarm_L1" : Bool AT %DB5059.DBX47.4, 500 ms
   "2925RS001A01F02.FP_EN.Alarm_L2" : Bool AT %DB5059.DBX47.5, 500 ms
   "2925RS001A01F02.FP_EN.Alarm_L3" : Bool AT %DB5059.DBX47.6, 500 ms
   "2925RS001A01F02.FP_EN.AlarmDelay_H3" : Bool AT %DB5059.DBX47.7, 500 ms
   "2925RS001A01F02.FP_EN.AlarmDelay_H2" : Bool AT %DB5059.DBX48.0, 500 ms
   "2925RS001A01F02.FP_EN.AlarmDelay_H1" : Bool AT %DB5059.DBX48.1, 500 ms
   "2925RS001A01F02.FP_EN.AlarmDelay_L1" : Bool AT %DB5059.DBX48.2, 500 ms
   "2925RS001A01F02.FP_EN.AlarmDelay_L2" : Bool AT %DB5059.DBX48.3, 500 ms
   "2925RS001A01F02.FP_EN.AlarmDelay_L3" : Bool AT %DB5059.DBX48.4, 500 ms
   "2925RS001A01F02.FP_EN.ROC_Warn" : Bool AT %DB5059.DBX48.5, 500 ms
   "2925RS001A01F02.FP_EN.U_Range_Warn" : Bool AT %DB5059.DBX48.6, 500 ms
   "2925RS001A01F02.FP_EN.O_Range_Warn" : Bool AT %DB5059.DBX48.7, 500 ms
   "2925RS001A01F02.trend_tag_name" : TextRef, internal   // Еденицы измерения При експорте из ECS через скрипт - заполняется автоматически, если теги копируются в ручную то требуется задатать свойство Text - имя тега для тренда
   "2925RS001A01F02.DQ.AL_H3" : Bool AT %DB5059.DBX16.0, 500 ms
   "2925RS001A01F02.DQ.AL_H2" : Bool AT %DB5059.DBX16.1, 500 ms
   "2925RS001A01F02.DQ.AL_H1" : Bool AT %DB5059.DBX16.2, 500 ms
   "2925RS001A01F02.DQ.AL_L1" : Bool AT %DB5059.DBX16.3, 500 ms
   "2925RS001A01F02.DQ.AL_L2" : Bool AT %DB5059.DBX16.4, 500 ms
   "2925RS001A01F02.DQ.AL_L3" : Bool AT %DB5059.DBX16.5, 500 ms
   "2925RS001A01F02.DQ.SIG_OK" : Bool AT %DB5059.DBX16.6, 500 ms
   "2925RS001A01F02.DQ.LIM_H2" : Bool AT %DB5059.DBX16.7, 500 ms
   "2925RS001A01F02.DQ.LIM_H1" : Bool AT %DB5059.DBX17.0, 500 ms
   "2925RS001A01F02.DQ.LIM_L1" : Bool AT %DB5059.DBX17.1, 500 ms
   "2925RS001A01F02.DQ.LIM_L2" : Bool AT %DB5059.DBX17.2, 500 ms
   "2925RS001A01F02.DQ.GR_P" : Bool AT %DB5059.DBX17.3, 500 ms
   "2925RS001A01F02.DQ.GR_N" : Bool AT %DB5059.DBX17.4, 500 ms
   "2925RS001A01F02.I.IN" : Real AT %DB5059.DBD2, 500 ms
   "2925RS001A01F02.I.SIG_TYPE" : Int AT %DB5059.DBW0, 500 ms
   "2925RS001A01F02.I.FI_BUS" : Byte AT %DB5059.DBB6, 500 ms
   "2925RS001A01F02.DI.U_RANGE" : Bool AT %DB5059.DBX7.0, 500 ms
   "2925RS001A01F02.DI.O_RANGE" : Bool AT %DB5059.DBX7.1, 500 ms
   "2925RS001A01F02.DI.SIG_FAULT" : Bool AT %DB5059.DBX7.2, 500 ms
   "2925RS001A01F02.DI.EnConfig" : Bool AT %DB5059.DBX7.3, 500 ms
   "2925RS001A01F02.DI.AEN" : Bool AT %DB5059.DBX7.4, 500 ms
   "2925RS001A01F02.DI.AL_SUPR" : Bool AT %DB5059.DBX7.5, 500 ms
   "2925RS001A01F02.Q.PV_NORM" : Real AT %DB5059.DBD8, 500 ms
   "2925RS001A01F02.Q.PV_SCAL" : Real AT %DB5059.DBD12, 500 ms
   "2925RS001A01F02.ParentInfo" : TextRef, internal   // Имя родителя для попап окна, вкладка инфо. При експорте из ECS через скрипт заполняется автоматически, если теги копируются в ручную то требуется в ручную задатать свойство Start Value

HMI tags "2925RS001A01F03"
   "2925RS001A01F03.MSW" : 52809b66-421d-457f-8884-6f7a49d4e247 AT %DB5060.DBX18.0, 500 ms
   "2925RS001A01F03.DefaultText" : TextRef, internal   // Заголовок POPUP окна. При експорте из ECS через скрипт заполняется автоматически, если теги копируются в ручную то требуется в ручную задатать свойство Start Value
   "2925RS001A01F03.BlockInfo" : Array [0..2] of Int AT %DB5060.DBX38.0, 500 ms
   "2925RS001A01F03.StatusWork" : Int AT %DB5060.DBW242, 500 ms
   "2925RS001A01F03.FP_PARAM.DampingTime" : Int AT %DB5060.DBW50, 500 ms
   "2925RS001A01F03.FP_PARAM.Force_Value" : Real AT %DB5060.DBD52, 500 ms
   "2925RS001A01F03.FP_PARAM.Scale_Min" : Real AT %DB5060.DBD56, 500 ms
   "2925RS001A01F03.FP_PARAM.Scale_Max" : Real AT %DB5060.DBD60, 500 ms
   "2925RS001A01F03.FP_PARAM.Gradient" : Real AT %DB5060.DBD64, 500 ms
   "2925RS001A01F03.FP_PARAM.Grad_Pos" : Real AT %DB5060.DBD68, 500 ms
   "2925RS001A01F03.FP_PARAM.Grad_Neg" : Real AT %DB5060.DBD72, 500 ms
   "2925RS001A01F03.FP_PARAM.Grad_X" : Real AT %DB5060.DBD76, 500 ms
   "2925RS001A01F03.FP_PARAM.Gradient_Time_Pre" : Int AT %DB5060.DBW80, 500 ms
   "2925RS001A01F03.FP_PARAM.Gradient_Time_ACC" : Int AT %DB5060.DBW82, 500 ms
   "2925RS001A01F03.FP_PARAM.Alarm_Hyst" : Real AT %DB5060.DBD84, 500 ms
   "2925RS001A01F03.FP_PARAM.AlarmLimit_H3" : Real AT %DB5060.DBD88, 500 ms
   "2925RS001A01F03.FP_PARAM.AlarmLimit_H2" : Real AT %DB5060.DBD92, 500 ms
   "2925RS001A01F03.FP_PARAM.AlarmLimit_H1" : Real AT %DB5060.DBD96, 500 ms
   "2925RS001A01F03.FP_PARAM.AlarmLimit_L1" : Real AT %DB5060.DBD100, 500 ms
   "2925RS001A01F03.FP_PARAM.AlarmLimit_L2" : Real AT %DB5060.DBD104, 500 ms
   "2925RS001A01F03.FP_PARAM.AlarmLimit_L3" : Real AT %DB5060.DBD108, 500 ms
   "2925RS001A01F03.FP_PARAM.AlarmDelay_H3_Pre" : Int AT %DB5060.DBW112, 500 ms
   "2925RS001A01F03.FP_PARAM.AlarmDelay_H3_Acc" : Int AT %DB5060.DBW114, 500 ms
   "2925RS001A01F03.FP_PARAM.AlarmDelay_H2_Pre" : Int AT %DB5060.DBW116, 500 ms
   "2925RS001A01F03.FP_PARAM.AlarmDelay_H2_Acc" : Int AT %DB5060.DBW118, 500 ms
   "2925RS001A01F03.FP_PARAM.AlarmDelay_H1_Pre" : Int AT %DB5060.DBW120, 500 ms
   "2925RS001A01F03.FP_PARAM.AlarmDelay_H1_Acc" : Int AT %DB5060.DBW122, 500 ms
   "2925RS001A01F03.FP_PARAM.AlarmDelay_L1_Pre" : Int AT %DB5060.DBW124, 500 ms
   "2925RS001A01F03.FP_PARAM.AlarmDelay_L1_Acc" : Int AT %DB5060.DBW126, 500 ms
   "2925RS001A01F03.FP_PARAM.AlarmDelay_L2_Pre" : Int AT %DB5060.DBW128, 500 ms
   "2925RS001A01F03.FP_PARAM.AlarmDelay_L2_Acc" : Int AT %DB5060.DBW130, 500 ms
   "2925RS001A01F03.FP_PARAM.AlarmDelay_L3_Pre" : Int AT %DB5060.DBW132, 500 ms
   "2925RS001A01F03.FP_PARAM.AlarmDelay_L3_Acc" : Int AT %DB5060.DBW134, 500 ms
   "2925RS001A01F03.FP_PARAM.OpenLoopDelay_Pre" : Int AT %DB5060.DBW136, 500 ms
   "2925RS001A01F03.FP_PARAM.OpenLoopDelay_Acc" : Int AT %DB5060.DBW138, 500 ms
   "2925RS001A01F03.FP_PARAM.OverRangeDelay_Pre" : Int AT %DB5060.DBW140, 500 ms
   "2925RS001A01F03.FP_PARAM.OverRangeDelay_Acc" : Int AT %DB5060.DBW142, 500 ms
   "2925RS001A01F03.FP_PARAM.AuxLimit_H2_Value" : Real AT %DB5060.DBD144, 500 ms
   "2925RS001A01F03.FP_PARAM.AuxLimit_H1_Value" : Real AT %DB5060.DBD148, 500 ms
   "2925RS001A01F03.FP_PARAM.AuxLimit_L2_Value" : Real AT %DB5060.DBD152, 500 ms
   "2925RS001A01F03.FP_PARAM.AuxLimit_L1_Value" : Real AT %DB5060.DBD156, 500 ms
   "2925RS001A01F03.Unit" : TextRef, internal   // Еденицы измерения При експорте из ECS через скрипт заполняется автоматически, если теги копируются в ручную то требуется задатать свойство Text
   "2925RS001A01F03.Decimals" : TextRef, internal   // Формат отображения При експорте из ECS через скрипт, заполняется автоматически. Если теги копируются в ручную то требуется задатать свойство Text s999999.9
   "2925RS001A01F03.FP_EN.Square" : Bool AT %DB5060.DBX46.0, 500 ms
   "2925RS001A01F03.FP_EN.SquareRoot" : Bool AT %DB5060.DBX46.1, 500 ms
   "2925RS001A01F03.FP_EN.ParentSupress" : Bool AT %DB5060.DBX46.2, 500 ms
   "2925RS001A01F03.FP_EN.ParentSupressUnit" : Bool AT %DB5060.DBX46.3, 500 ms
   "2925RS001A01F03.FP_EN.Force" : Bool AT %DB5060.DBX46.4, 500 ms
   "2925RS001A01F03.FP_EN.Damping" : Bool AT %DB5060.DBX46.5, 500 ms
   "2925RS001A01F03.FP_EN.Gradient_Pos" : Bool AT %DB5060.DBX46.6, 500 ms
   "2925RS001A01F03.FP_EN.Gradient_Neg" : Bool AT %DB5060.DBX46.7, 500 ms
   "2925RS001A01F03.FP_EN.Hysteresis" : Bool AT %DB5060.DBX47.0, 500 ms
   "2925RS001A01F03.FP_EN.Alarm_H3" : Bool AT %DB5060.DBX47.1, 500 ms
   "2925RS001A01F03.FP_EN.Alarm_H2" : Bool AT %DB5060.DBX47.2, 500 ms
   "2925RS001A01F03.FP_EN.Alarm_H1" : Bool AT %DB5060.DBX47.3, 500 ms
   "2925RS001A01F03.FP_EN.Alarm_L1" : Bool AT %DB5060.DBX47.4, 500 ms
   "2925RS001A01F03.FP_EN.Alarm_L2" : Bool AT %DB5060.DBX47.5, 500 ms
   "2925RS001A01F03.FP_EN.Alarm_L3" : Bool AT %DB5060.DBX47.6, 500 ms
   "2925RS001A01F03.FP_EN.AlarmDelay_H3" : Bool AT %DB5060.DBX47.7, 500 ms
   "2925RS001A01F03.FP_EN.AlarmDelay_H2" : Bool AT %DB5060.DBX48.0, 500 ms
   "2925RS001A01F03.FP_EN.AlarmDelay_H1" : Bool AT %DB5060.DBX48.1, 500 ms
   "2925RS001A01F03.FP_EN.AlarmDelay_L1" : Bool AT %DB5060.DBX48.2, 500 ms
   "2925RS001A01F03.FP_EN.AlarmDelay_L2" : Bool AT %DB5060.DBX48.3, 500 ms
   "2925RS001A01F03.FP_EN.AlarmDelay_L3" : Bool AT %DB5060.DBX48.4, 500 ms
   "2925RS001A01F03.FP_EN.ROC_Warn" : Bool AT %DB5060.DBX48.5, 500 ms
   "2925RS001A01F03.FP_EN.U_Range_Warn" : Bool AT %DB5060.DBX48.6, 500 ms
   "2925RS001A01F03.FP_EN.O_Range_Warn" : Bool AT %DB5060.DBX48.7, 500 ms
   "2925RS001A01F03.trend_tag_name" : TextRef, internal   // Еденицы измерения При експорте из ECS через скрипт - заполняется автоматически, если теги копируются в ручную то требуется задатать свойство Text - имя тега для тренда
   "2925RS001A01F03.DQ.AL_H3" : Bool AT %DB5060.DBX16.0, 500 ms
   "2925RS001A01F03.DQ.AL_H2" : Bool AT %DB5060.DBX16.1, 500 ms
   "2925RS001A01F03.DQ.AL_H1" : Bool AT %DB5060.DBX16.2, 500 ms
   "2925RS001A01F03.DQ.AL_L1" : Bool AT %DB5060.DBX16.3, 500 ms
   "2925RS001A01F03.DQ.AL_L2" : Bool AT %DB5060.DBX16.4, 500 ms
   "2925RS001A01F03.DQ.AL_L3" : Bool AT %DB5060.DBX16.5, 500 ms
   "2925RS001A01F03.DQ.SIG_OK" : Bool AT %DB5060.DBX16.6, 500 ms
   "2925RS001A01F03.DQ.LIM_H2" : Bool AT %DB5060.DBX16.7, 500 ms
   "2925RS001A01F03.DQ.LIM_H1" : Bool AT %DB5060.DBX17.0, 500 ms
   "2925RS001A01F03.DQ.LIM_L1" : Bool AT %DB5060.DBX17.1, 500 ms
   "2925RS001A01F03.DQ.LIM_L2" : Bool AT %DB5060.DBX17.2, 500 ms
   "2925RS001A01F03.DQ.GR_P" : Bool AT %DB5060.DBX17.3, 500 ms
   "2925RS001A01F03.DQ.GR_N" : Bool AT %DB5060.DBX17.4, 500 ms
   "2925RS001A01F03.I.IN" : Real AT %DB5060.DBD2, 500 ms
   "2925RS001A01F03.I.SIG_TYPE" : Int AT %DB5060.DBW0, 500 ms
   "2925RS001A01F03.I.FI_BUS" : Byte AT %DB5060.DBB6, 500 ms
   "2925RS001A01F03.DI.U_RANGE" : Bool AT %DB5060.DBX7.0, 500 ms
   "2925RS001A01F03.DI.O_RANGE" : Bool AT %DB5060.DBX7.1, 500 ms
   "2925RS001A01F03.DI.SIG_FAULT" : Bool AT %DB5060.DBX7.2, 500 ms
   "2925RS001A01F03.DI.EnConfig" : Bool AT %DB5060.DBX7.3, 500 ms
   "2925RS001A01F03.DI.AEN" : Bool AT %DB5060.DBX7.4, 500 ms
   "2925RS001A01F03.DI.AL_SUPR" : Bool AT %DB5060.DBX7.5, 500 ms
   "2925RS001A01F03.Q.PV_NORM" : Real AT %DB5060.DBD8, 500 ms
   "2925RS001A01F03.Q.PV_SCAL" : Real AT %DB5060.DBD12, 500 ms
   "2925RS001A01F03.ParentInfo" : TextRef, internal   // Имя родителя для попап окна, вкладка инфо. При експорте из ECS через скрипт заполняется автоматически, если теги копируются в ручную то требуется в ручную задатать свойство Start Value

HMI tags "2925RS001A01F04"
   "2925RS001A01F04.MSW" : 52809b66-421d-457f-8884-6f7a49d4e247 AT %DB5061.DBX18.0, 500 ms
   "2925RS001A01F04.DefaultText" : TextRef, internal   // Заголовок POPUP окна. При експорте из ECS через скрипт заполняется автоматически, если теги копируются в ручную то требуется в ручную задатать свойство Start Value
   "2925RS001A01F04.BlockInfo" : Array [0..2] of Int AT %DB5061.DBX38.0, 500 ms
   "2925RS001A01F04.StatusWork" : Int AT %DB5061.DBW242, 500 ms
   "2925RS001A01F04.FP_PARAM.DampingTime" : Int AT %DB5061.DBW50, 500 ms
   "2925RS001A01F04.FP_PARAM.Force_Value" : Real AT %DB5061.DBD52, 500 ms
   "2925RS001A01F04.FP_PARAM.Scale_Min" : Real AT %DB5061.DBD56, 500 ms
   "2925RS001A01F04.FP_PARAM.Scale_Max" : Real AT %DB5061.DBD60, 500 ms
   "2925RS001A01F04.FP_PARAM.Gradient" : Real AT %DB5061.DBD64, 500 ms
   "2925RS001A01F04.FP_PARAM.Grad_Pos" : Real AT %DB5061.DBD68, 500 ms
   "2925RS001A01F04.FP_PARAM.Grad_Neg" : Real AT %DB5061.DBD72, 500 ms
   "2925RS001A01F04.FP_PARAM.Grad_X" : Real AT %DB5061.DBD76, 500 ms
   "2925RS001A01F04.FP_PARAM.Gradient_Time_Pre" : Int AT %DB5061.DBW80, 500 ms
   "2925RS001A01F04.FP_PARAM.Gradient_Time_ACC" : Int AT %DB5061.DBW82, 500 ms
   "2925RS001A01F04.FP_PARAM.Alarm_Hyst" : Real AT %DB5061.DBD84, 500 ms
   "2925RS001A01F04.FP_PARAM.AlarmLimit_H3" : Real AT %DB5061.DBD88, 500 ms
   "2925RS001A01F04.FP_PARAM.AlarmLimit_H2" : Real AT %DB5061.DBD92, 500 ms
   "2925RS001A01F04.FP_PARAM.AlarmLimit_H1" : Real AT %DB5061.DBD96, 500 ms
   "2925RS001A01F04.FP_PARAM.AlarmLimit_L1" : Real AT %DB5061.DBD100, 500 ms
   "2925RS001A01F04.FP_PARAM.AlarmLimit_L2" : Real AT %DB5061.DBD104, 500 ms
   "2925RS001A01F04.FP_PARAM.AlarmLimit_L3" : Real AT %DB5061.DBD108, 500 ms
   "2925RS001A01F04.FP_PARAM.AlarmDelay_H3_Pre" : Int AT %DB5061.DBW112, 500 ms
   "2925RS001A01F04.FP_PARAM.AlarmDelay_H3_Acc" : Int AT %DB5061.DBW114, 500 ms
   "2925RS001A01F04.FP_PARAM.AlarmDelay_H2_Pre" : Int AT %DB5061.DBW116, 500 ms
   "2925RS001A01F04.FP_PARAM.AlarmDelay_H2_Acc" : Int AT %DB5061.DBW118, 500 ms
   "2925RS001A01F04.FP_PARAM.AlarmDelay_H1_Pre" : Int AT %DB5061.DBW120, 500 ms
   "2925RS001A01F04.FP_PARAM.AlarmDelay_H1_Acc" : Int AT %DB5061.DBW122, 500 ms
   "2925RS001A01F04.FP_PARAM.AlarmDelay_L1_Pre" : Int AT %DB5061.DBW124, 500 ms
   "2925RS001A01F04.FP_PARAM.AlarmDelay_L1_Acc" : Int AT %DB5061.DBW126, 500 ms
   "2925RS001A01F04.FP_PARAM.AlarmDelay_L2_Pre" : Int AT %DB5061.DBW128, 500 ms
   "2925RS001A01F04.FP_PARAM.AlarmDelay_L2_Acc" : Int AT %DB5061.DBW130, 500 ms
   "2925RS001A01F04.FP_PARAM.AlarmDelay_L3_Pre" : Int AT %DB5061.DBW132, 500 ms
   "2925RS001A01F04.FP_PARAM.AlarmDelay_L3_Acc" : Int AT %DB5061.DBW134, 500 ms
   "2925RS001A01F04.FP_PARAM.OpenLoopDelay_Pre" : Int AT %DB5061.DBW136, 500 ms
   "2925RS001A01F04.FP_PARAM.OpenLoopDelay_Acc" : Int AT %DB5061.DBW138, 500 ms
   "2925RS001A01F04.FP_PARAM.OverRangeDelay_Pre" : Int AT %DB5061.DBW140, 500 ms
   "2925RS001A01F04.FP_PARAM.OverRangeDelay_Acc" : Int AT %DB5061.DBW142, 500 ms
   "2925RS001A01F04.FP_PARAM.AuxLimit_H2_Value" : Real AT %DB5061.DBD144, 500 ms
   "2925RS001A01F04.FP_PARAM.AuxLimit_H1_Value" : Real AT %DB5061.DBD148, 500 ms
   "2925RS001A01F04.FP_PARAM.AuxLimit_L2_Value" : Real AT %DB5061.DBD152, 500 ms
   "2925RS001A01F04.FP_PARAM.AuxLimit_L1_Value" : Real AT %DB5061.DBD156, 500 ms
   "2925RS001A01F04.Unit" : TextRef, internal   // Еденицы измерения При експорте из ECS через скрипт заполняется автоматически, если теги копируются в ручную то требуется задатать свойство Text
   "2925RS001A01F04.Decimals" : TextRef, internal   // Формат отображения При експорте из ECS через скрипт, заполняется автоматически. Если теги копируются в ручную то требуется задатать свойство Text s999999.9
   "2925RS001A01F04.FP_EN.Square" : Bool AT %DB5061.DBX46.0, 500 ms
   "2925RS001A01F04.FP_EN.SquareRoot" : Bool AT %DB5061.DBX46.1, 500 ms
   "2925RS001A01F04.FP_EN.ParentSupress" : Bool AT %DB5061.DBX46.2, 500 ms
   "2925RS001A01F04.FP_EN.ParentSupressUnit" : Bool AT %DB5061.DBX46.3, 500 ms
   "2925RS001A01F04.FP_EN.Force" : Bool AT %DB5061.DBX46.4, 500 ms
   "2925RS001A01F04.FP_EN.Damping" : Bool AT %DB5061.DBX46.5, 500 ms
   "2925RS001A01F04.FP_EN.Gradient_Pos" : Bool AT %DB5061.DBX46.6, 500 ms
   "2925RS001A01F04.FP_EN.Gradient_Neg" : Bool AT %DB5061.DBX46.7, 500 ms
   "2925RS001A01F04.FP_EN.Hysteresis" : Bool AT %DB5061.DBX47.0, 500 ms
   "2925RS001A01F04.FP_EN.Alarm_H3" : Bool AT %DB5061.DBX47.1, 500 ms
   "2925RS001A01F04.FP_EN.Alarm_H2" : Bool AT %DB5061.DBX47.2, 500 ms
   "2925RS001A01F04.FP_EN.Alarm_H1" : Bool AT %DB5061.DBX47.3, 500 ms
   "2925RS001A01F04.FP_EN.Alarm_L1" : Bool AT %DB5061.DBX47.4, 500 ms
   "2925RS001A01F04.FP_EN.Alarm_L2" : Bool AT %DB5061.DBX47.5, 500 ms
   "2925RS001A01F04.FP_EN.Alarm_L3" : Bool AT %DB5061.DBX47.6, 500 ms
   "2925RS001A01F04.FP_EN.AlarmDelay_H3" : Bool AT %DB5061.DBX47.7, 500 ms
   "2925RS001A01F04.FP_EN.AlarmDelay_H2" : Bool AT %DB5061.DBX48.0, 500 ms
   "2925RS001A01F04.FP_EN.AlarmDelay_H1" : Bool AT %DB5061.DBX48.1, 500 ms
   "2925RS001A01F04.FP_EN.AlarmDelay_L1" : Bool AT %DB5061.DBX48.2, 500 ms
   "2925RS001A01F04.FP_EN.AlarmDelay_L2" : Bool AT %DB5061.DBX48.3, 500 ms
   "2925RS001A01F04.FP_EN.AlarmDelay_L3" : Bool AT %DB5061.DBX48.4, 500 ms
   "2925RS001A01F04.FP_EN.ROC_Warn" : Bool AT %DB5061.DBX48.5, 500 ms
   "2925RS001A01F04.FP_EN.U_Range_Warn" : Bool AT %DB5061.DBX48.6, 500 ms
   "2925RS001A01F04.FP_EN.O_Range_Warn" : Bool AT %DB5061.DBX48.7, 500 ms
   "2925RS001A01F04.trend_tag_name" : TextRef, internal   // Еденицы измерения При експорте из ECS через скрипт - заполняется автоматически, если теги копируются в ручную то требуется задатать свойство Text - имя тега для тренда
   "2925RS001A01F04.DQ.AL_H3" : Bool AT %DB5061.DBX16.0, 500 ms
   "2925RS001A01F04.DQ.AL_H2" : Bool AT %DB5061.DBX16.1, 500 ms
   "2925RS001A01F04.DQ.AL_H1" : Bool AT %DB5061.DBX16.2, 500 ms
   "2925RS001A01F04.DQ.AL_L1" : Bool AT %DB5061.DBX16.3, 500 ms
   "2925RS001A01F04.DQ.AL_L2" : Bool AT %DB5061.DBX16.4, 500 ms
   "2925RS001A01F04.DQ.AL_L3" : Bool AT %DB5061.DBX16.5, 500 ms
   "2925RS001A01F04.DQ.SIG_OK" : Bool AT %DB5061.DBX16.6, 500 ms
   "2925RS001A01F04.DQ.LIM_H2" : Bool AT %DB5061.DBX16.7, 500 ms
   "2925RS001A01F04.DQ.LIM_H1" : Bool AT %DB5061.DBX17.0, 500 ms
   "2925RS001A01F04.DQ.LIM_L1" : Bool AT %DB5061.DBX17.1, 500 ms
   "2925RS001A01F04.DQ.LIM_L2" : Bool AT %DB5061.DBX17.2, 500 ms
   "2925RS001A01F04.DQ.GR_P" : Bool AT %DB5061.DBX17.3, 500 ms
   "2925RS001A01F04.DQ.GR_N" : Bool AT %DB5061.DBX17.4, 500 ms
   "2925RS001A01F04.I.IN" : Real AT %DB5061.DBD2, 500 ms
   "2925RS001A01F04.I.SIG_TYPE" : Int AT %DB5061.DBW0, 500 ms
   "2925RS001A01F04.I.FI_BUS" : Byte AT %DB5061.DBB6, 500 ms
   "2925RS001A01F04.DI.U_RANGE" : Bool AT %DB5061.DBX7.0, 500 ms
   "2925RS001A01F04.DI.O_RANGE" : Bool AT %DB5061.DBX7.1, 500 ms
   "2925RS001A01F04.DI.SIG_FAULT" : Bool AT %DB5061.DBX7.2, 500 ms
   "2925RS001A01F04.DI.EnConfig" : Bool AT %DB5061.DBX7.3, 500 ms
   "2925RS001A01F04.DI.AEN" : Bool AT %DB5061.DBX7.4, 500 ms
   "2925RS001A01F04.DI.AL_SUPR" : Bool AT %DB5061.DBX7.5, 500 ms
   "2925RS001A01F04.Q.PV_NORM" : Real AT %DB5061.DBD8, 500 ms
   "2925RS001A01F04.Q.PV_SCAL" : Real AT %DB5061.DBD12, 500 ms
   "2925RS001A01F04.ParentInfo" : TextRef, internal   // Имя родителя для попап окна, вкладка инфо. При експорте из ECS через скрипт заполняется автоматически, если теги копируются в ручную то требуется в ручную задатать свойство Start Value

HMI tags "2925RS001A01F05"
   "2925RS001A01F05.MSW" : 52809b66-421d-457f-8884-6f7a49d4e247 AT %DB5062.DBX18.0, 500 ms
   "2925RS001A01F05.DefaultText" : TextRef, internal   // Заголовок POPUP окна. При експорте из ECS через скрипт заполняется автоматически, если теги копируются в ручную то требуется в ручную задатать свойство Start Value
   "2925RS001A01F05.BlockInfo" : Array [0..2] of Int AT %DB5062.DBX38.0, 500 ms
   "2925RS001A01F05.StatusWork" : Int AT %DB5062.DBW242, 500 ms
   "2925RS001A01F05.FP_PARAM.DampingTime" : Int AT %DB5062.DBW50, 500 ms
   "2925RS001A01F05.FP_PARAM.Force_Value" : Real AT %DB5062.DBD52, 500 ms
   "2925RS001A01F05.FP_PARAM.Scale_Min" : Real AT %DB5062.DBD56, 500 ms
   "2925RS001A01F05.FP_PARAM.Scale_Max" : Real AT %DB5062.DBD60, 500 ms
   "2925RS001A01F05.FP_PARAM.Gradient" : Real AT %DB5062.DBD64, 500 ms
   "2925RS001A01F05.FP_PARAM.Grad_Pos" : Real AT %DB5062.DBD68, 500 ms
   "2925RS001A01F05.FP_PARAM.Grad_Neg" : Real AT %DB5062.DBD72, 500 ms
   "2925RS001A01F05.FP_PARAM.Grad_X" : Real AT %DB5062.DBD76, 500 ms
   "2925RS001A01F05.FP_PARAM.Gradient_Time_Pre" : Int AT %DB5062.DBW80, 500 ms
   "2925RS001A01F05.FP_PARAM.Gradient_Time_ACC" : Int AT %DB5062.DBW82, 500 ms
   "2925RS001A01F05.FP_PARAM.Alarm_Hyst" : Real AT %DB5062.DBD84, 500 ms
   "2925RS001A01F05.FP_PARAM.AlarmLimit_H3" : Real AT %DB5062.DBD88, 500 ms
   "2925RS001A01F05.FP_PARAM.AlarmLimit_H2" : Real AT %DB5062.DBD92, 500 ms
   "2925RS001A01F05.FP_PARAM.AlarmLimit_H1" : Real AT %DB5062.DBD96, 500 ms
   "2925RS001A01F05.FP_PARAM.AlarmLimit_L1" : Real AT %DB5062.DBD100, 500 ms
   "2925RS001A01F05.FP_PARAM.AlarmLimit_L2" : Real AT %DB5062.DBD104, 500 ms
   "2925RS001A01F05.FP_PARAM.AlarmLimit_L3" : Real AT %DB5062.DBD108, 500 ms
   "2925RS001A01F05.FP_PARAM.AlarmDelay_H3_Pre" : Int AT %DB5062.DBW112, 500 ms
   "2925RS001A01F05.FP_PARAM.AlarmDelay_H3_Acc" : Int AT %DB5062.DBW114, 500 ms
   "2925RS001A01F05.FP_PARAM.AlarmDelay_H2_Pre" : Int AT %DB5062.DBW116, 500 ms
   "2925RS001A01F05.FP_PARAM.AlarmDelay_H2_Acc" : Int AT %DB5062.DBW118, 500 ms
   "2925RS001A01F05.FP_PARAM.AlarmDelay_H1_Pre" : Int AT %DB5062.DBW120, 500 ms
   "2925RS001A01F05.FP_PARAM.AlarmDelay_H1_Acc" : Int AT %DB5062.DBW122, 500 ms
   "2925RS001A01F05.FP_PARAM.AlarmDelay_L1_Pre" : Int AT %DB5062.DBW124, 500 ms
   "2925RS001A01F05.FP_PARAM.AlarmDelay_L1_Acc" : Int AT %DB5062.DBW126, 500 ms
   "2925RS001A01F05.FP_PARAM.AlarmDelay_L2_Pre" : Int AT %DB5062.DBW128, 500 ms
   "2925RS001A01F05.FP_PARAM.AlarmDelay_L2_Acc" : Int AT %DB5062.DBW130, 500 ms
   "2925RS001A01F05.FP_PARAM.AlarmDelay_L3_Pre" : Int AT %DB5062.DBW132, 500 ms
   "2925RS001A01F05.FP_PARAM.AlarmDelay_L3_Acc" : Int AT %DB5062.DBW134, 500 ms
   "2925RS001A01F05.FP_PARAM.OpenLoopDelay_Pre" : Int AT %DB5062.DBW136, 500 ms
   "2925RS001A01F05.FP_PARAM.OpenLoopDelay_Acc" : Int AT %DB5062.DBW138, 500 ms
   "2925RS001A01F05.FP_PARAM.OverRangeDelay_Pre" : Int AT %DB5062.DBW140, 500 ms
   "2925RS001A01F05.FP_PARAM.OverRangeDelay_Acc" : Int AT %DB5062.DBW142, 500 ms
   "2925RS001A01F05.FP_PARAM.AuxLimit_H2_Value" : Real AT %DB5062.DBD144, 500 ms
   "2925RS001A01F05.FP_PARAM.AuxLimit_H1_Value" : Real AT %DB5062.DBD148, 500 ms
   "2925RS001A01F05.FP_PARAM.AuxLimit_L2_Value" : Real AT %DB5062.DBD152, 500 ms
   "2925RS001A01F05.FP_PARAM.AuxLimit_L1_Value" : Real AT %DB5062.DBD156, 500 ms
   "2925RS001A01F05.Unit" : TextRef, internal   // Еденицы измерения При експорте из ECS через скрипт заполняется автоматически, если теги копируются в ручную то требуется задатать свойство Text
   "2925RS001A01F05.Decimals" : TextRef, internal   // Формат отображения При експорте из ECS через скрипт, заполняется автоматически. Если теги копируются в ручную то требуется задатать свойство Text s999999.9
   "2925RS001A01F05.FP_EN.Square" : Bool AT %DB5062.DBX46.0, 500 ms
   "2925RS001A01F05.FP_EN.SquareRoot" : Bool AT %DB5062.DBX46.1, 500 ms
   "2925RS001A01F05.FP_EN.ParentSupress" : Bool AT %DB5062.DBX46.2, 500 ms
   "2925RS001A01F05.FP_EN.ParentSupressUnit" : Bool AT %DB5062.DBX46.3, 500 ms
   "2925RS001A01F05.FP_EN.Force" : Bool AT %DB5062.DBX46.4, 500 ms
   "2925RS001A01F05.FP_EN.Damping" : Bool AT %DB5062.DBX46.5, 500 ms
   "2925RS001A01F05.FP_EN.Gradient_Pos" : Bool AT %DB5062.DBX46.6, 500 ms
   "2925RS001A01F05.FP_EN.Gradient_Neg" : Bool AT %DB5062.DBX46.7, 500 ms
   "2925RS001A01F05.FP_EN.Hysteresis" : Bool AT %DB5062.DBX47.0, 500 ms
   "2925RS001A01F05.FP_EN.Alarm_H3" : Bool AT %DB5062.DBX47.1, 500 ms
   "2925RS001A01F05.FP_EN.Alarm_H2" : Bool AT %DB5062.DBX47.2, 500 ms
   "2925RS001A01F05.FP_EN.Alarm_H1" : Bool AT %DB5062.DBX47.3, 500 ms
   "2925RS001A01F05.FP_EN.Alarm_L1" : Bool AT %DB5062.DBX47.4, 500 ms
   "2925RS001A01F05.FP_EN.Alarm_L2" : Bool AT %DB5062.DBX47.5, 500 ms
   "2925RS001A01F05.FP_EN.Alarm_L3" : Bool AT %DB5062.DBX47.6, 500 ms
   "2925RS001A01F05.FP_EN.AlarmDelay_H3" : Bool AT %DB5062.DBX47.7, 500 ms
   "2925RS001A01F05.FP_EN.AlarmDelay_H2" : Bool AT %DB5062.DBX48.0, 500 ms
   "2925RS001A01F05.FP_EN.AlarmDelay_H1" : Bool AT %DB5062.DBX48.1, 500 ms
   "2925RS001A01F05.FP_EN.AlarmDelay_L1" : Bool AT %DB5062.DBX48.2, 500 ms
   "2925RS001A01F05.FP_EN.AlarmDelay_L2" : Bool AT %DB5062.DBX48.3, 500 ms
   "2925RS001A01F05.FP_EN.AlarmDelay_L3" : Bool AT %DB5062.DBX48.4, 500 ms
   "2925RS001A01F05.FP_EN.ROC_Warn" : Bool AT %DB5062.DBX48.5, 500 ms
   "2925RS001A01F05.FP_EN.U_Range_Warn" : Bool AT %DB5062.DBX48.6, 500 ms
   "2925RS001A01F05.FP_EN.O_Range_Warn" : Bool AT %DB5062.DBX48.7, 500 ms
   "2925RS001A01F05.trend_tag_name" : TextRef, internal   // Еденицы измерения При експорте из ECS через скрипт - заполняется автоматически, если теги копируются в ручную то требуется задатать свойство Text - имя тега для тренда
   "2925RS001A01F05.DQ.AL_H3" : Bool AT %DB5062.DBX16.0, 500 ms
   "2925RS001A01F05.DQ.AL_H2" : Bool AT %DB5062.DBX16.1, 500 ms
   "2925RS001A01F05.DQ.AL_H1" : Bool AT %DB5062.DBX16.2, 500 ms
   "2925RS001A01F05.DQ.AL_L1" : Bool AT %DB5062.DBX16.3, 500 ms
   "2925RS001A01F05.DQ.AL_L2" : Bool AT %DB5062.DBX16.4, 500 ms
   "2925RS001A01F05.DQ.AL_L3" : Bool AT %DB5062.DBX16.5, 500 ms
   "2925RS001A01F05.DQ.SIG_OK" : Bool AT %DB5062.DBX16.6, 500 ms
   "2925RS001A01F05.DQ.LIM_H2" : Bool AT %DB5062.DBX16.7, 500 ms
   "2925RS001A01F05.DQ.LIM_H1" : Bool AT %DB5062.DBX17.0, 500 ms
   "2925RS001A01F05.DQ.LIM_L1" : Bool AT %DB5062.DBX17.1, 500 ms
   "2925RS001A01F05.DQ.LIM_L2" : Bool AT %DB5062.DBX17.2, 500 ms
   "2925RS001A01F05.DQ.GR_P" : Bool AT %DB5062.DBX17.3, 500 ms
   "2925RS001A01F05.DQ.GR_N" : Bool AT %DB5062.DBX17.4, 500 ms
   "2925RS001A01F05.I.IN" : Real AT %DB5062.DBD2, 500 ms
   "2925RS001A01F05.I.SIG_TYPE" : Int AT %DB5062.DBW0, 500 ms
   "2925RS001A01F05.I.FI_BUS" : Byte AT %DB5062.DBB6, 500 ms
   "2925RS001A01F05.DI.U_RANGE" : Bool AT %DB5062.DBX7.0, 500 ms
   "2925RS001A01F05.DI.O_RANGE" : Bool AT %DB5062.DBX7.1, 500 ms
   "2925RS001A01F05.DI.SIG_FAULT" : Bool AT %DB5062.DBX7.2, 500 ms
   "2925RS001A01F05.DI.EnConfig" : Bool AT %DB5062.DBX7.3, 500 ms
   "2925RS001A01F05.DI.AEN" : Bool AT %DB5062.DBX7.4, 500 ms
   "2925RS001A01F05.DI.AL_SUPR" : Bool AT %DB5062.DBX7.5, 500 ms
   "2925RS001A01F05.Q.PV_NORM" : Real AT %DB5062.DBD8, 500 ms
   "2925RS001A01F05.Q.PV_SCAL" : Real AT %DB5062.DBD12, 500 ms
   "2925RS001A01F05.ParentInfo" : TextRef, internal   // Имя родителя для попап окна, вкладка инфо. При експорте из ECS через скрипт заполняется автоматически, если теги копируются в ручную то требуется в ручную задатать свойство Start Value

HMI tags "2925RS001A01F06"
   "2925RS001A01F06.MSW" : 52809b66-421d-457f-8884-6f7a49d4e247 AT %DB5063.DBX18.0, 500 ms
   "2925RS001A01F06.DefaultText" : TextRef, internal   // Заголовок POPUP окна. При експорте из ECS через скрипт заполняется автоматически, если теги копируются в ручную то требуется в ручную задатать свойство Start Value
   "2925RS001A01F06.BlockInfo" : Array [0..2] of Int AT %DB5063.DBX38.0, 500 ms
   "2925RS001A01F06.StatusWork" : Int AT %DB5063.DBW242, 500 ms
   "2925RS001A01F06.FP_PARAM.DampingTime" : Int AT %DB5063.DBW50, 500 ms
   "2925RS001A01F06.FP_PARAM.Force_Value" : Real AT %DB5063.DBD52, 500 ms
   "2925RS001A01F06.FP_PARAM.Scale_Min" : Real AT %DB5063.DBD56, 500 ms
   "2925RS001A01F06.FP_PARAM.Scale_Max" : Real AT %DB5063.DBD60, 500 ms
   "2925RS001A01F06.FP_PARAM.Gradient" : Real AT %DB5063.DBD64, 500 ms
   "2925RS001A01F06.FP_PARAM.Grad_Pos" : Real AT %DB5063.DBD68, 500 ms
   "2925RS001A01F06.FP_PARAM.Grad_Neg" : Real AT %DB5063.DBD72, 500 ms
   "2925RS001A01F06.FP_PARAM.Grad_X" : Real AT %DB5063.DBD76, 500 ms
   "2925RS001A01F06.FP_PARAM.Gradient_Time_Pre" : Int AT %DB5063.DBW80, 500 ms
   "2925RS001A01F06.FP_PARAM.Gradient_Time_ACC" : Int AT %DB5063.DBW82, 500 ms
   "2925RS001A01F06.FP_PARAM.Alarm_Hyst" : Real AT %DB5063.DBD84, 500 ms
   "2925RS001A01F06.FP_PARAM.AlarmLimit_H3" : Real AT %DB5063.DBD88, 500 ms
   "2925RS001A01F06.FP_PARAM.AlarmLimit_H2" : Real AT %DB5063.DBD92, 500 ms
   "2925RS001A01F06.FP_PARAM.AlarmLimit_H1" : Real AT %DB5063.DBD96, 500 ms
   "2925RS001A01F06.FP_PARAM.AlarmLimit_L1" : Real AT %DB5063.DBD100, 500 ms
   "2925RS001A01F06.FP_PARAM.AlarmLimit_L2" : Real AT %DB5063.DBD104, 500 ms
   "2925RS001A01F06.FP_PARAM.AlarmLimit_L3" : Real AT %DB5063.DBD108, 500 ms
   "2925RS001A01F06.FP_PARAM.AlarmDelay_H3_Pre" : Int AT %DB5063.DBW112, 500 ms
   "2925RS001A01F06.FP_PARAM.AlarmDelay_H3_Acc" : Int AT %DB5063.DBW114, 500 ms
   "2925RS001A01F06.FP_PARAM.AlarmDelay_H2_Pre" : Int AT %DB5063.DBW116, 500 ms
   "2925RS001A01F06.FP_PARAM.AlarmDelay_H2_Acc" : Int AT %DB5063.DBW118, 500 ms
   "2925RS001A01F06.FP_PARAM.AlarmDelay_H1_Pre" : Int AT %DB5063.DBW120, 500 ms
   "2925RS001A01F06.FP_PARAM.AlarmDelay_H1_Acc" : Int AT %DB5063.DBW122, 500 ms
   "2925RS001A01F06.FP_PARAM.AlarmDelay_L1_Pre" : Int AT %DB5063.DBW124, 500 ms
   "2925RS001A01F06.FP_PARAM.AlarmDelay_L1_Acc" : Int AT %DB5063.DBW126, 500 ms
   "2925RS001A01F06.FP_PARAM.AlarmDelay_L2_Pre" : Int AT %DB5063.DBW128, 500 ms
   "2925RS001A01F06.FP_PARAM.AlarmDelay_L2_Acc" : Int AT %DB5063.DBW130, 500 ms
   "2925RS001A01F06.FP_PARAM.AlarmDelay_L3_Pre" : Int AT %DB5063.DBW132, 500 ms
   "2925RS001A01F06.FP_PARAM.AlarmDelay_L3_Acc" : Int AT %DB5063.DBW134, 500 ms
   "2925RS001A01F06.FP_PARAM.OpenLoopDelay_Pre" : Int AT %DB5063.DBW136, 500 ms
   "2925RS001A01F06.FP_PARAM.OpenLoopDelay_Acc" : Int AT %DB5063.DBW138, 500 ms
   "2925RS001A01F06.FP_PARAM.OverRangeDelay_Pre" : Int AT %DB5063.DBW140, 500 ms
   "2925RS001A01F06.FP_PARAM.OverRangeDelay_Acc" : Int AT %DB5063.DBW142, 500 ms
   "2925RS001A01F06.FP_PARAM.AuxLimit_H2_Value" : Real AT %DB5063.DBD144, 500 ms
   "2925RS001A01F06.FP_PARAM.AuxLimit_H1_Value" : Real AT %DB5063.DBD148, 500 ms
   "2925RS001A01F06.FP_PARAM.AuxLimit_L2_Value" : Real AT %DB5063.DBD152, 500 ms
   "2925RS001A01F06.FP_PARAM.AuxLimit_L1_Value" : Real AT %DB5063.DBD156, 500 ms
   "2925RS001A01F06.Unit" : TextRef, internal   // Еденицы измерения При експорте из ECS через скрипт заполняется автоматически, если теги копируются в ручную то требуется задатать свойство Text
   "2925RS001A01F06.Decimals" : TextRef, internal   // Формат отображения При експорте из ECS через скрипт, заполняется автоматически. Если теги копируются в ручную то требуется задатать свойство Text s999999.9
   "2925RS001A01F06.FP_EN.Square" : Bool AT %DB5063.DBX46.0, 500 ms
   "2925RS001A01F06.FP_EN.SquareRoot" : Bool AT %DB5063.DBX46.1, 500 ms
   "2925RS001A01F06.FP_EN.ParentSupress" : Bool AT %DB5063.DBX46.2, 500 ms
   "2925RS001A01F06.FP_EN.ParentSupressUnit" : Bool AT %DB5063.DBX46.3, 500 ms
   "2925RS001A01F06.FP_EN.Force" : Bool AT %DB5063.DBX46.4, 500 ms
   "2925RS001A01F06.FP_EN.Damping" : Bool AT %DB5063.DBX46.5, 500 ms
   "2925RS001A01F06.FP_EN.Gradient_Pos" : Bool AT %DB5063.DBX46.6, 500 ms
   "2925RS001A01F06.FP_EN.Gradient_Neg" : Bool AT %DB5063.DBX46.7, 500 ms
   "2925RS001A01F06.FP_EN.Hysteresis" : Bool AT %DB5063.DBX47.0, 500 ms
   "2925RS001A01F06.FP_EN.Alarm_H3" : Bool AT %DB5063.DBX47.1, 500 ms
   "2925RS001A01F06.FP_EN.Alarm_H2" : Bool AT %DB5063.DBX47.2, 500 ms
   "2925RS001A01F06.FP_EN.Alarm_H1" : Bool AT %DB5063.DBX47.3, 500 ms
   "2925RS001A01F06.FP_EN.Alarm_L1" : Bool AT %DB5063.DBX47.4, 500 ms
   "2925RS001A01F06.FP_EN.Alarm_L2" : Bool AT %DB5063.DBX47.5, 500 ms
   "2925RS001A01F06.FP_EN.Alarm_L3" : Bool AT %DB5063.DBX47.6, 500 ms
   "2925RS001A01F06.FP_EN.AlarmDelay_H3" : Bool AT %DB5063.DBX47.7, 500 ms
   "2925RS001A01F06.FP_EN.AlarmDelay_H2" : Bool AT %DB5063.DBX48.0, 500 ms
   "2925RS001A01F06.FP_EN.AlarmDelay_H1" : Bool AT %DB5063.DBX48.1, 500 ms
   "2925RS001A01F06.FP_EN.AlarmDelay_L1" : Bool AT %DB5063.DBX48.2, 500 ms
   "2925RS001A01F06.FP_EN.AlarmDelay_L2" : Bool AT %DB5063.DBX48.3, 500 ms
   "2925RS001A01F06.FP_EN.AlarmDelay_L3" : Bool AT %DB5063.DBX48.4, 500 ms
   "2925RS001A01F06.FP_EN.ROC_Warn" : Bool AT %DB5063.DBX48.5, 500 ms
   "2925RS001A01F06.FP_EN.U_Range_Warn" : Bool AT %DB5063.DBX48.6, 500 ms
   "2925RS001A01F06.FP_EN.O_Range_Warn" : Bool AT %DB5063.DBX48.7, 500 ms
   "2925RS001A01F06.trend_tag_name" : TextRef, internal   // Еденицы измерения При експорте из ECS через скрипт - заполняется автоматически, если теги копируются в ручную то требуется задатать свойство Text - имя тега для тренда
   "2925RS001A01F06.DQ.AL_H3" : Bool AT %DB5063.DBX16.0, 500 ms
   "2925RS001A01F06.DQ.AL_H2" : Bool AT %DB5063.DBX16.1, 500 ms
   "2925RS001A01F06.DQ.AL_H1" : Bool AT %DB5063.DBX16.2, 500 ms
   "2925RS001A01F06.DQ.AL_L1" : Bool AT %DB5063.DBX16.3, 500 ms
   "2925RS001A01F06.DQ.AL_L2" : Bool AT %DB5063.DBX16.4, 500 ms
   "2925RS001A01F06.DQ.AL_L3" : Bool AT %DB5063.DBX16.5, 500 ms
   "2925RS001A01F06.DQ.SIG_OK" : Bool AT %DB5063.DBX16.6, 500 ms
   "2925RS001A01F06.DQ.LIM_H2" : Bool AT %DB5063.DBX16.7, 500 ms
   "2925RS001A01F06.DQ.LIM_H1" : Bool AT %DB5063.DBX17.0, 500 ms
   "2925RS001A01F06.DQ.LIM_L1" : Bool AT %DB5063.DBX17.1, 500 ms
   "2925RS001A01F06.DQ.LIM_L2" : Bool AT %DB5063.DBX17.2, 500 ms
   "2925RS001A01F06.DQ.GR_P" : Bool AT %DB5063.DBX17.3, 500 ms
   "2925RS001A01F06.DQ.GR_N" : Bool AT %DB5063.DBX17.4, 500 ms
   "2925RS001A01F06.I.IN" : Real AT %DB5063.DBD2, 500 ms
   "2925RS001A01F06.I.SIG_TYPE" : Int AT %DB5063.DBW0, 500 ms
   "2925RS001A01F06.I.FI_BUS" : Byte AT %DB5063.DBB6, 500 ms
   "2925RS001A01F06.DI.U_RANGE" : Bool AT %DB5063.DBX7.0, 500 ms
   "2925RS001A01F06.DI.O_RANGE" : Bool AT %DB5063.DBX7.1, 500 ms
   "2925RS001A01F06.DI.SIG_FAULT" : Bool AT %DB5063.DBX7.2, 500 ms
   "2925RS001A01F06.DI.EnConfig" : Bool AT %DB5063.DBX7.3, 500 ms
   "2925RS001A01F06.DI.AEN" : Bool AT %DB5063.DBX7.4, 500 ms
   "2925RS001A01F06.DI.AL_SUPR" : Bool AT %DB5063.DBX7.5, 500 ms
   "2925RS001A01F06.Q.PV_NORM" : Real AT %DB5063.DBD8, 500 ms
   "2925RS001A01F06.Q.PV_SCAL" : Real AT %DB5063.DBD12, 500 ms
   "2925RS001A01F06.ParentInfo" : TextRef, internal   // Имя родителя для попап окна, вкладка инфо. При експорте из ECS через скрипт заполняется автоматически, если теги копируются в ручную то требуется в ручную задатать свойство Start Value

HMI tags "2925RS001A01F07"
   "2925RS001A01F07.MSW" : 52809b66-421d-457f-8884-6f7a49d4e247 AT %DB5064.DBX18.0, 500 ms
   "2925RS001A01F07.DefaultText" : TextRef, internal   // Заголовок POPUP окна. При експорте из ECS через скрипт заполняется автоматически, если теги копируются в ручную то требуется в ручную задатать свойство Start Value
   "2925RS001A01F07.BlockInfo" : Array [0..2] of Int AT %DB5064.DBX38.0, 500 ms
   "2925RS001A01F07.StatusWork" : Int AT %DB5064.DBW242, 500 ms
   "2925RS001A01F07.FP_PARAM.DampingTime" : Int AT %DB5064.DBW50, 500 ms
   "2925RS001A01F07.FP_PARAM.Force_Value" : Real AT %DB5064.DBD52, 500 ms
   "2925RS001A01F07.FP_PARAM.Scale_Min" : Real AT %DB5064.DBD56, 500 ms
   "2925RS001A01F07.FP_PARAM.Scale_Max" : Real AT %DB5064.DBD60, 500 ms
   "2925RS001A01F07.FP_PARAM.Gradient" : Real AT %DB5064.DBD64, 500 ms
   "2925RS001A01F07.FP_PARAM.Grad_Pos" : Real AT %DB5064.DBD68, 500 ms
   "2925RS001A01F07.FP_PARAM.Grad_Neg" : Real AT %DB5064.DBD72, 500 ms
   "2925RS001A01F07.FP_PARAM.Grad_X" : Real AT %DB5064.DBD76, 500 ms
   "2925RS001A01F07.FP_PARAM.Gradient_Time_Pre" : Int AT %DB5064.DBW80, 500 ms
   "2925RS001A01F07.FP_PARAM.Gradient_Time_ACC" : Int AT %DB5064.DBW82, 500 ms
   "2925RS001A01F07.FP_PARAM.Alarm_Hyst" : Real AT %DB5064.DBD84, 500 ms
   "2925RS001A01F07.FP_PARAM.AlarmLimit_H3" : Real AT %DB5064.DBD88, 500 ms
   "2925RS001A01F07.FP_PARAM.AlarmLimit_H2" : Real AT %DB5064.DBD92, 500 ms
   "2925RS001A01F07.FP_PARAM.AlarmLimit_H1" : Real AT %DB5064.DBD96, 500 ms
   "2925RS001A01F07.FP_PARAM.AlarmLimit_L1" : Real AT %DB5064.DBD100, 500 ms
   "2925RS001A01F07.FP_PARAM.AlarmLimit_L2" : Real AT %DB5064.DBD104, 500 ms
   "2925RS001A01F07.FP_PARAM.AlarmLimit_L3" : Real AT %DB5064.DBD108, 500 ms
   "2925RS001A01F07.FP_PARAM.AlarmDelay_H3_Pre" : Int AT %DB5064.DBW112, 500 ms
   "2925RS001A01F07.FP_PARAM.AlarmDelay_H3_Acc" : Int AT %DB5064.DBW114, 500 ms
   "2925RS001A01F07.FP_PARAM.AlarmDelay_H2_Pre" : Int AT %DB5064.DBW116, 500 ms
   "2925RS001A01F07.FP_PARAM.AlarmDelay_H2_Acc" : Int AT %DB5064.DBW118, 500 ms
   "2925RS001A01F07.FP_PARAM.AlarmDelay_H1_Pre" : Int AT %DB5064.DBW120, 500 ms
   "2925RS001A01F07.FP_PARAM.AlarmDelay_H1_Acc" : Int AT %DB5064.DBW122, 500 ms
   "2925RS001A01F07.FP_PARAM.AlarmDelay_L1_Pre" : Int AT %DB5064.DBW124, 500 ms
   "2925RS001A01F07.FP_PARAM.AlarmDelay_L1_Acc" : Int AT %DB5064.DBW126, 500 ms
   "2925RS001A01F07.FP_PARAM.AlarmDelay_L2_Pre" : Int AT %DB5064.DBW128, 500 ms
   "2925RS001A01F07.FP_PARAM.AlarmDelay_L2_Acc" : Int AT %DB5064.DBW130, 500 ms
   "2925RS001A01F07.FP_PARAM.AlarmDelay_L3_Pre" : Int AT %DB5064.DBW132, 500 ms
   "2925RS001A01F07.FP_PARAM.AlarmDelay_L3_Acc" : Int AT %DB5064.DBW134, 500 ms
   "2925RS001A01F07.FP_PARAM.OpenLoopDelay_Pre" : Int AT %DB5064.DBW136, 500 ms
   "2925RS001A01F07.FP_PARAM.OpenLoopDelay_Acc" : Int AT %DB5064.DBW138, 500 ms
   "2925RS001A01F07.FP_PARAM.OverRangeDelay_Pre" : Int AT %DB5064.DBW140, 500 ms
   "2925RS001A01F07.FP_PARAM.OverRangeDelay_Acc" : Int AT %DB5064.DBW142, 500 ms
   "2925RS001A01F07.FP_PARAM.AuxLimit_H2_Value" : Real AT %DB5064.DBD144, 500 ms
   "2925RS001A01F07.FP_PARAM.AuxLimit_H1_Value" : Real AT %DB5064.DBD148, 500 ms
   "2925RS001A01F07.FP_PARAM.AuxLimit_L2_Value" : Real AT %DB5064.DBD152, 500 ms
   "2925RS001A01F07.FP_PARAM.AuxLimit_L1_Value" : Real AT %DB5064.DBD156, 500 ms
   "2925RS001A01F07.Unit" : TextRef, internal   // Еденицы измерения При експорте из ECS через скрипт заполняется автоматически, если теги копируются в ручную то требуется задатать свойство Text
   "2925RS001A01F07.Decimals" : TextRef, internal   // Формат отображения При експорте из ECS через скрипт, заполняется автоматически. Если теги копируются в ручную то требуется задатать свойство Text s999999.9
   "2925RS001A01F07.FP_EN.Square" : Bool AT %DB5064.DBX46.0, 500 ms
   "2925RS001A01F07.FP_EN.SquareRoot" : Bool AT %DB5064.DBX46.1, 500 ms
   "2925RS001A01F07.FP_EN.ParentSupress" : Bool AT %DB5064.DBX46.2, 500 ms
   "2925RS001A01F07.FP_EN.ParentSupressUnit" : Bool AT %DB5064.DBX46.3, 500 ms
   "2925RS001A01F07.FP_EN.Force" : Bool AT %DB5064.DBX46.4, 500 ms
   "2925RS001A01F07.FP_EN.Damping" : Bool AT %DB5064.DBX46.5, 500 ms
   "2925RS001A01F07.FP_EN.Gradient_Pos" : Bool AT %DB5064.DBX46.6, 500 ms
   "2925RS001A01F07.FP_EN.Gradient_Neg" : Bool AT %DB5064.DBX46.7, 500 ms
   "2925RS001A01F07.FP_EN.Hysteresis" : Bool AT %DB5064.DBX47.0, 500 ms
   "2925RS001A01F07.FP_EN.Alarm_H3" : Bool AT %DB5064.DBX47.1, 500 ms
   "2925RS001A01F07.FP_EN.Alarm_H2" : Bool AT %DB5064.DBX47.2, 500 ms
   "2925RS001A01F07.FP_EN.Alarm_H1" : Bool AT %DB5064.DBX47.3, 500 ms
   "2925RS001A01F07.FP_EN.Alarm_L1" : Bool AT %DB5064.DBX47.4, 500 ms
   "2925RS001A01F07.FP_EN.Alarm_L2" : Bool AT %DB5064.DBX47.5, 500 ms
   "2925RS001A01F07.FP_EN.Alarm_L3" : Bool AT %DB5064.DBX47.6, 500 ms
   "2925RS001A01F07.FP_EN.AlarmDelay_H3" : Bool AT %DB5064.DBX47.7, 500 ms
   "2925RS001A01F07.FP_EN.AlarmDelay_H2" : Bool AT %DB5064.DBX48.0, 500 ms
   "2925RS001A01F07.FP_EN.AlarmDelay_H1" : Bool AT %DB5064.DBX48.1, 500 ms
   "2925RS001A01F07.FP_EN.AlarmDelay_L1" : Bool AT %DB5064.DBX48.2, 500 ms
   "2925RS001A01F07.FP_EN.AlarmDelay_L2" : Bool AT %DB5064.DBX48.3, 500 ms
   "2925RS001A01F07.FP_EN.AlarmDelay_L3" : Bool AT %DB5064.DBX48.4, 500 ms
   "2925RS001A01F07.FP_EN.ROC_Warn" : Bool AT %DB5064.DBX48.5, 500 ms
   "2925RS001A01F07.FP_EN.U_Range_Warn" : Bool AT %DB5064.DBX48.6, 500 ms
   "2925RS001A01F07.FP_EN.O_Range_Warn" : Bool AT %DB5064.DBX48.7, 500 ms
   "2925RS001A01F07.trend_tag_name" : TextRef, internal   // Еденицы измерения При експорте из ECS через скрипт - заполняется автоматически, если теги копируются в ручную то требуется задатать свойство Text - имя тега для тренда
   "2925RS001A01F07.DQ.AL_H3" : Bool AT %DB5064.DBX16.0, 500 ms
   "2925RS001A01F07.DQ.AL_H2" : Bool AT %DB5064.DBX16.1, 500 ms
   "2925RS001A01F07.DQ.AL_H1" : Bool AT %DB5064.DBX16.2, 500 ms
   "2925RS001A01F07.DQ.AL_L1" : Bool AT %DB5064.DBX16.3, 500 ms
   "2925RS001A01F07.DQ.AL_L2" : Bool AT %DB5064.DBX16.4, 500 ms
   "2925RS001A01F07.DQ.AL_L3" : Bool AT %DB5064.DBX16.5, 500 ms
   "2925RS001A01F07.DQ.SIG_OK" : Bool AT %DB5064.DBX16.6, 500 ms
   "2925RS001A01F07.DQ.LIM_H2" : Bool AT %DB5064.DBX16.7, 500 ms
   "2925RS001A01F07.DQ.LIM_H1" : Bool AT %DB5064.DBX17.0, 500 ms
   "2925RS001A01F07.DQ.LIM_L1" : Bool AT %DB5064.DBX17.1, 500 ms
   "2925RS001A01F07.DQ.LIM_L2" : Bool AT %DB5064.DBX17.2, 500 ms
   "2925RS001A01F07.DQ.GR_P" : Bool AT %DB5064.DBX17.3, 500 ms
   "2925RS001A01F07.DQ.GR_N" : Bool AT %DB5064.DBX17.4, 500 ms
   "2925RS001A01F07.I.IN" : Real AT %DB5064.DBD2, 500 ms
   "2925RS001A01F07.I.SIG_TYPE" : Int AT %DB5064.DBW0, 500 ms
   "2925RS001A01F07.I.FI_BUS" : Byte AT %DB5064.DBB6, 500 ms
   "2925RS001A01F07.DI.U_RANGE" : Bool AT %DB5064.DBX7.0, 500 ms
   "2925RS001A01F07.DI.O_RANGE" : Bool AT %DB5064.DBX7.1, 500 ms
   "2925RS001A01F07.DI.SIG_FAULT" : Bool AT %DB5064.DBX7.2, 500 ms
   "2925RS001A01F07.DI.EnConfig" : Bool AT %DB5064.DBX7.3, 500 ms
   "2925RS001A01F07.DI.AEN" : Bool AT %DB5064.DBX7.4, 500 ms
   "2925RS001A01F07.DI.AL_SUPR" : Bool AT %DB5064.DBX7.5, 500 ms
   "2925RS001A01F07.Q.PV_NORM" : Real AT %DB5064.DBD8, 500 ms
   "2925RS001A01F07.Q.PV_SCAL" : Real AT %DB5064.DBD12, 500 ms
   "2925RS001A01F07.ParentInfo" : TextRef, internal   // Имя родителя для попап окна, вкладка инфо. При експорте из ECS через скрипт заполняется автоматически, если теги копируются в ручную то требуется в ручную задатать свойство Start Value

HMI tags "2925RS001A01L01"
   "2925RS001A01L01.MSW" : 52809b66-421d-457f-8884-6f7a49d4e247 AT %DB5065.DBX18.0, 500 ms
   "2925RS001A01L01.DefaultText" : TextRef, internal   // Заголовок POPUP окна. При експорте из ECS через скрипт заполняется автоматически, если теги копируются в ручную то требуется в ручную задатать свойство Start Value
   "2925RS001A01L01.BlockInfo" : Array [0..2] of Int AT %DB5065.DBX38.0, 500 ms
   "2925RS001A01L01.StatusWork" : Int AT %DB5065.DBW242, 500 ms
   "2925RS001A01L01.FP_PARAM.DampingTime" : Int AT %DB5065.DBW50, 500 ms
   "2925RS001A01L01.FP_PARAM.Force_Value" : Real AT %DB5065.DBD52, 500 ms
   "2925RS001A01L01.FP_PARAM.Scale_Min" : Real AT %DB5065.DBD56, 500 ms
   "2925RS001A01L01.FP_PARAM.Scale_Max" : Real AT %DB5065.DBD60, 500 ms
   "2925RS001A01L01.FP_PARAM.Gradient" : Real AT %DB5065.DBD64, 500 ms
   "2925RS001A01L01.FP_PARAM.Grad_Pos" : Real AT %DB5065.DBD68, 500 ms
   "2925RS001A01L01.FP_PARAM.Grad_Neg" : Real AT %DB5065.DBD72, 500 ms
   "2925RS001A01L01.FP_PARAM.Grad_X" : Real AT %DB5065.DBD76, 500 ms
   "2925RS001A01L01.FP_PARAM.Gradient_Time_Pre" : Int AT %DB5065.DBW80, 500 ms
   "2925RS001A01L01.FP_PARAM.Gradient_Time_ACC" : Int AT %DB5065.DBW82, 500 ms
   "2925RS001A01L01.FP_PARAM.Alarm_Hyst" : Real AT %DB5065.DBD84, 500 ms
   "2925RS001A01L01.FP_PARAM.AlarmLimit_H3" : Real AT %DB5065.DBD88, 500 ms
   "2925RS001A01L01.FP_PARAM.AlarmLimit_H2" : Real AT %DB5065.DBD92, 500 ms
   "2925RS001A01L01.FP_PARAM.AlarmLimit_H1" : Real AT %DB5065.DBD96, 500 ms
   "2925RS001A01L01.FP_PARAM.AlarmLimit_L1" : Real AT %DB5065.DBD100, 500 ms
   "2925RS001A01L01.FP_PARAM.AlarmLimit_L2" : Real AT %DB5065.DBD104, 500 ms
   "2925RS001A01L01.FP_PARAM.AlarmLimit_L3" : Real AT %DB5065.DBD108, 500 ms
   "2925RS001A01L01.FP_PARAM.AlarmDelay_H3_Pre" : Int AT %DB5065.DBW112, 500 ms
   "2925RS001A01L01.FP_PARAM.AlarmDelay_H3_Acc" : Int AT %DB5065.DBW114, 500 ms
   "2925RS001A01L01.FP_PARAM.AlarmDelay_H2_Pre" : Int AT %DB5065.DBW116, 500 ms
   "2925RS001A01L01.FP_PARAM.AlarmDelay_H2_Acc" : Int AT %DB5065.DBW118, 500 ms
   "2925RS001A01L01.FP_PARAM.AlarmDelay_H1_Pre" : Int AT %DB5065.DBW120, 500 ms
   "2925RS001A01L01.FP_PARAM.AlarmDelay_H1_Acc" : Int AT %DB5065.DBW122, 500 ms
   "2925RS001A01L01.FP_PARAM.AlarmDelay_L1_Pre" : Int AT %DB5065.DBW124, 500 ms
   "2925RS001A01L01.FP_PARAM.AlarmDelay_L1_Acc" : Int AT %DB5065.DBW126, 500 ms
   "2925RS001A01L01.FP_PARAM.AlarmDelay_L2_Pre" : Int AT %DB5065.DBW128, 500 ms
   "2925RS001A01L01.FP_PARAM.AlarmDelay_L2_Acc" : Int AT %DB5065.DBW130, 500 ms
   "2925RS001A01L01.FP_PARAM.AlarmDelay_L3_Pre" : Int AT %DB5065.DBW132, 500 ms
   "2925RS001A01L01.FP_PARAM.AlarmDelay_L3_Acc" : Int AT %DB5065.DBW134, 500 ms
   "2925RS001A01L01.FP_PARAM.OpenLoopDelay_Pre" : Int AT %DB5065.DBW136, 500 ms
   "2925RS001A01L01.FP_PARAM.OpenLoopDelay_Acc" : Int AT %DB5065.DBW138, 500 ms
   "2925RS001A01L01.FP_PARAM.OverRangeDelay_Pre" : Int AT %DB5065.DBW140, 500 ms
   "2925RS001A01L01.FP_PARAM.OverRangeDelay_Acc" : Int AT %DB5065.DBW142, 500 ms
   "2925RS001A01L01.FP_PARAM.AuxLimit_H2_Value" : Real AT %DB5065.DBD144, 500 ms
   "2925RS001A01L01.FP_PARAM.AuxLimit_H1_Value" : Real AT %DB5065.DBD148, 500 ms
   "2925RS001A01L01.FP_PARAM.AuxLimit_L2_Value" : Real AT %DB5065.DBD152, 500 ms
   "2925RS001A01L01.FP_PARAM.AuxLimit_L1_Value" : Real AT %DB5065.DBD156, 500 ms
   "2925RS001A01L01.Unit" : TextRef, internal   // Еденицы измерения При експорте из ECS через скрипт заполняется автоматически, если теги копируются в ручную то требуется задатать свойство Text
   "2925RS001A01L01.Decimals" : TextRef, internal   // Формат отображения При експорте из ECS через скрипт, заполняется автоматически. Если теги копируются в ручную то требуется задатать свойство Text s999999.9
   "2925RS001A01L01.FP_EN.Square" : Bool AT %DB5065.DBX46.0, 500 ms
   "2925RS001A01L01.FP_EN.SquareRoot" : Bool AT %DB5065.DBX46.1, 500 ms
   "2925RS001A01L01.FP_EN.ParentSupress" : Bool AT %DB5065.DBX46.2, 500 ms
   "2925RS001A01L01.FP_EN.ParentSupressUnit" : Bool AT %DB5065.DBX46.3, 500 ms
   "2925RS001A01L01.FP_EN.Force" : Bool AT %DB5065.DBX46.4, 500 ms
   "2925RS001A01L01.FP_EN.Damping" : Bool AT %DB5065.DBX46.5, 500 ms
   "2925RS001A01L01.FP_EN.Gradient_Pos" : Bool AT %DB5065.DBX46.6, 500 ms
   "2925RS001A01L01.FP_EN.Gradient_Neg" : Bool AT %DB5065.DBX46.7, 500 ms
   "2925RS001A01L01.FP_EN.Hysteresis" : Bool AT %DB5065.DBX47.0, 500 ms
   "2925RS001A01L01.FP_EN.Alarm_H3" : Bool AT %DB5065.DBX47.1, 500 ms
   "2925RS001A01L01.FP_EN.Alarm_H2" : Bool AT %DB5065.DBX47.2, 500 ms
   "2925RS001A01L01.FP_EN.Alarm_H1" : Bool AT %DB5065.DBX47.3, 500 ms
   "2925RS001A01L01.FP_EN.Alarm_L1" : Bool AT %DB5065.DBX47.4, 500 ms
   "2925RS001A01L01.FP_EN.Alarm_L2" : Bool AT %DB5065.DBX47.5, 500 ms
   "2925RS001A01L01.FP_EN.Alarm_L3" : Bool AT %DB5065.DBX47.6, 500 ms
   "2925RS001A01L01.FP_EN.AlarmDelay_H3" : Bool AT %DB5065.DBX47.7, 500 ms
   "2925RS001A01L01.FP_EN.AlarmDelay_H2" : Bool AT %DB5065.DBX48.0, 500 ms
   "2925RS001A01L01.FP_EN.AlarmDelay_H1" : Bool AT %DB5065.DBX48.1, 500 ms
   "2925RS001A01L01.FP_EN.AlarmDelay_L1" : Bool AT %DB5065.DBX48.2, 500 ms
   "2925RS001A01L01.FP_EN.AlarmDelay_L2" : Bool AT %DB5065.DBX48.3, 500 ms
   "2925RS001A01L01.FP_EN.AlarmDelay_L3" : Bool AT %DB5065.DBX48.4, 500 ms
   "2925RS001A01L01.FP_EN.ROC_Warn" : Bool AT %DB5065.DBX48.5, 500 ms
   "2925RS001A01L01.FP_EN.U_Range_Warn" : Bool AT %DB5065.DBX48.6, 500 ms
   "2925RS001A01L01.FP_EN.O_Range_Warn" : Bool AT %DB5065.DBX48.7, 500 ms
   "2925RS001A01L01.trend_tag_name" : TextRef, internal   // Еденицы измерения При експорте из ECS через скрипт - заполняется автоматически, если теги копируются в ручную то требуется задатать свойство Text - имя тега для тренда
   "2925RS001A01L01.DQ.AL_H3" : Bool AT %DB5065.DBX16.0, 500 ms
   "2925RS001A01L01.DQ.AL_H2" : Bool AT %DB5065.DBX16.1, 500 ms
   "2925RS001A01L01.DQ.AL_H1" : Bool AT %DB5065.DBX16.2, 500 ms
   "2925RS001A01L01.DQ.AL_L1" : Bool AT %DB5065.DBX16.3, 500 ms
   "2925RS001A01L01.DQ.AL_L2" : Bool AT %DB5065.DBX16.4, 500 ms
   "2925RS001A01L01.DQ.AL_L3" : Bool AT %DB5065.DBX16.5, 500 ms
   "2925RS001A01L01.DQ.SIG_OK" : Bool AT %DB5065.DBX16.6, 500 ms
   "2925RS001A01L01.DQ.LIM_H2" : Bool AT %DB5065.DBX16.7, 500 ms
   "2925RS001A01L01.DQ.LIM_H1" : Bool AT %DB5065.DBX17.0, 500 ms
   "2925RS001A01L01.DQ.LIM_L1" : Bool AT %DB5065.DBX17.1, 500 ms
   "2925RS001A01L01.DQ.LIM_L2" : Bool AT %DB5065.DBX17.2, 500 ms
   "2925RS001A01L01.DQ.GR_P" : Bool AT %DB5065.DBX17.3, 500 ms
   "2925RS001A01L01.DQ.GR_N" : Bool AT %DB5065.DBX17.4, 500 ms
   "2925RS001A01L01.I.IN" : Real AT %DB5065.DBD2, 500 ms
   "2925RS001A01L01.I.SIG_TYPE" : Int AT %DB5065.DBW0, 500 ms
   "2925RS001A01L01.I.FI_BUS" : Byte AT %DB5065.DBB6, 500 ms
   "2925RS001A01L01.DI.U_RANGE" : Bool AT %DB5065.DBX7.0, 500 ms
   "2925RS001A01L01.DI.O_RANGE" : Bool AT %DB5065.DBX7.1, 500 ms
   "2925RS001A01L01.DI.SIG_FAULT" : Bool AT %DB5065.DBX7.2, 500 ms
   "2925RS001A01L01.DI.EnConfig" : Bool AT %DB5065.DBX7.3, 500 ms
   "2925RS001A01L01.DI.AEN" : Bool AT %DB5065.DBX7.4, 500 ms
   "2925RS001A01L01.DI.AL_SUPR" : Bool AT %DB5065.DBX7.5, 500 ms
   "2925RS001A01L01.Q.PV_NORM" : Real AT %DB5065.DBD8, 500 ms
   "2925RS001A01L01.Q.PV_SCAL" : Real AT %DB5065.DBD12, 500 ms
   "2925RS001A01L01.ParentInfo" : TextRef, internal   // Имя родителя для попап окна, вкладка инфо. При експорте из ECS через скрипт заполняется автоматически, если теги копируются в ручную то требуется в ручную задатать свойство Start Value

